  [779] = {x=22.893, y=-17.965, rx=-180, rz=-141.93, shoulder=lefty, elbow=epositive, wrist=wpositive, fatherId=fReference[0]}
  [780] = {x=24.131, y=-18.934, rx=180, rz=-141.938, shoulder=lefty, elbow=epositive, wrist=wpositive, fatherId=fReference[0]}
  [781] = {x=25.369, y=-19.904, rx=-180, rz=-141.947, shoulder=lefty, elbow=epositive, wrist=wpositive, fatherId=fReference[0]}
  [782] = {x=26.607, y=-20.873, rx=-180, rz=-141.956, shoulder=lefty, elbow=epositive, wrist=wpositive, fatherId=fReference[0]}
  [783] = {x=27.846, y=-21.842, rx=-180, rz=-141.965, shoulder=lefty, elbow=epositive, wrist=wpositive, fatherId=fReference[0]}
  [784] = {x=29.084, y=-22.811, rx=-180, rz=-141.975, shoulder=lefty, elbow=epositive, wrist=wpositive, fatherId=fReference[0]}
  [785] = {x=30.323, y=-23.779, rx=180, rz=-141.986, shoulder=lefty, elbow=epositive, wrist=wpositive, fatherId=fReference[0]}
  [786] = {x=31.561, y=-24.748, rx=-180, rz=-141.996, shoulder=lefty, elbow=epositive, wrist=wpositive, fatherId=fReference[0]}
  [787] = {x=32.8, y=-25.716, rx=-180, rz=-142.008, shoulder=lefty, elbow=epositive, wrist=wpositive, fatherId=fReference[0]}
  [788] = {x=34.039, y=-26.683, rx=-180, rz=-142.019, shoulder=lefty, elbow=epositive, wrist=wpositive, fatherId=fReference[0]}
  [789] = {x=35.278, y=-27.651, rx=-180, rz=-142.031, shoulder=lefty, elbow=epositive, wrist=wpositive, fatherId=fReference[0]}
  [790] = {x=36.517, y=-28.618, rx=-180, rz=-142.044, shoulder=lefty, elbow=epositive, wrist=wpositive, fatherId=fReference[0]}
  [791] = {x=37.757, y=-29.585, rx=180, rz=-142.057, shoulder=lefty, elbow=epositive, wrist=wpositive, fatherId=fReference[0]}
  [792] = {x=38.996, y=-30.551, rx=180, rz=-142.07, shoulder=lefty, elbow=epositive, wrist=wpositive, fatherId=fReference[0]}
  [793] = {x=40.236, y=-31.517, rx=180, rz=-142.084, shoulder=lefty, elbow=epositive, wrist=wpositive, fatherId=fReference[0]}
  [794] = {x=41.476, y=-32.483, rx=180, rz=-142.098, shoulder=lefty, elbow=epositive, wrist=wpositive, fatherId=fReference[0]}
  [795] = {x=42.715, y=-33.448, rx=180, rz=-142.113, shoulder=lefty, elbow=epositive, wrist=wpositive, fatherId=fReference[0]}
  [796] = {x=43.956, y=-34.413, rx=-180, rz=-142.128, shoulder=lefty, elbow=epositive, wrist=wpositive, fatherId=fReference[0]}
  [797] = {x=45.196, y=-35.377, rx=180, rz=-142.143, shoulder=lefty, elbow=epositive, wrist=wpositive, fatherId=fReference[0]}
  [798] = {x=46.436, y=-36.342, rx=-180, rz=-142.159, shoulder=lefty, elbow=epositive, wrist=wpositive, fatherId=fReference[0]}
  [799] = {x=47.677, y=-37.305, rx=180, rz=-142.175, shoulder=lefty, elbow=epositive, wrist=wpositive, fatherId=fReference[0]}
  [800] = {x=48.917, y=-38.269, rx=-180, rz=-142.192, shoulder=lefty, elbow=epositive, wrist=wpositive, fatherId=fReference[0]}
  [801] = {x=50.158, y=-39.231, rx=-180, rz=-142.209, shoulder=lefty, elbow=epositive, wrist=wpositive, fatherId=fReference[0]}
  [802] = {x=51.399, y=-40.194, rx=-180, rz=-142.227, shoulder=lefty, elbow=epositive, wrist=wpositive, fatherId=fReference[0]}
  [803] = {x=52.641, y=-41.156, rx=-180, rz=-142.245, shoulder=lefty, elbow=epositive, wrist=wpositive, fatherId=fReference[0]}
  [804] = {x=53.882, y=-42.117, rx=-180, rz=-142.263, shoulder=lefty, elbow=epositive, wrist=wpositive, fatherId=fReference[0]}
  [805] = {x=55.124, y=-43.078, rx=-180, rz=-142.282, shoulder=lefty, elbow=epositive, wrist=wpositive, fatherId=fReference[0]}
  [806] = {x=56.366, y=-44.038, rx=-180, rz=-142.302, shoulder=lefty, elbow=epositive, wrist=wpositive, fatherId=fReference[0]}
  [807] = {x=57.608, y=-44.998, rx=-180, rz=-142.321, shoulder=lefty, elbow=epositive, wrist=wpositive, fatherId=fReference[0]}
  [808] = {x=58.85, y=-45.958, rx=-180, rz=-142.342, shoulder=lefty, elbow=epositive, wrist=wpositive, fatherId=fReference[0]}
  [809] = {x=60.092, y=-46.916, rx=-180, rz=-142.362, shoulder=lefty, elbow=epositive, wrist=wpositive, fatherId=fReference[0]}
  [810] = {x=61.335, y=-47.875, rx=-180, rz=-142.383, shoulder=lefty, elbow=epositive, wrist=wpositive, fatherId=fReference[0]}
  [811] = {x=62.578, y=-48.832, rx=180, rz=-142.405, shoulder=lefty, elbow=epositive, wrist=wpositive, fatherId=fReference[0]}
  [812] = {x=63.821, y=-49.79, rx=-180, rz=-142.427, shoulder=lefty, elbow=epositive, wrist=wpositive, fatherId=fReference[0]}
  [813] = {x=65.064, y=-50.746, rx=180, rz=-142.449, shoulder=lefty, elbow=epositive, wrist=wpositive, fatherId=fReference[0]}
  [814] = {x=66.308, y=-51.702, rx=-180, rz=-142.472, shoulder=lefty, elbow=epositive, wrist=wpositive, fatherId=fReference[0]}
  [815] = {x=67.551, y=-52.657, rx=180, rz=-142.496, shoulder=lefty, elbow=epositive, wrist=wpositive, fatherId=fReference[0]}
  [816] = {x=68.795, y=-53.612, rx=180, rz=-142.519, shoulder=lefty, elbow=epositive, wrist=wpositive, fatherId=fReference[0]}
  [817] = {x=70.04, y=-54.566, rx=180, rz=-142.543, shoulder=lefty, elbow=epositive, wrist=wpositive, fatherId=fReference[0]}
  [818] = {x=71.284, y=-55.519, rx=-180, rz=-142.568, shoulder=lefty, elbow=epositive, wrist=wpositive, fatherId=fReference[0]}
  [819] = {x=72.529, y=-56.472, rx=-180, rz=-142.593, shoulder=lefty, elbow=epositive, wrist=wpositive, fatherId=fReference[0]}
  [820] = {x=73.774, y=-57.424, rx=-180, rz=-142.619, shoulder=lefty, elbow=epositive, wrist=wpositive, fatherId=fReference[0]}
  [821] = {x=75.019, y=-58.376, rx=180, rz=-142.645, shoulder=lefty, elbow=epositive, wrist=wpositive, fatherId=fReference[0]}
  [822] = {x=76.264, y=-59.326, rx=180, rz=-142.671, shoulder=lefty, elbow=epositive, wrist=wpositive, fatherId=fReference[0]}
  [823] = {x=77.51, y=-60.276, rx=180, rz=-142.698, shoulder=lefty, elbow=epositive, wrist=wpositive, fatherId=fReference[0]}
  [824] = {x=78.756, y=-61.226, rx=-180, rz=-142.725, shoulder=lefty, elbow=epositive, wrist=wpositive, fatherId=fReference[0]}
  [825] = {x=80.002, y=-62.174, rx=-180, rz=-142.753, shoulder=lefty, elbow=epositive, wrist=wpositive, fatherId=fReference[0]}
  [826] = {x=81.249, y=-63.122, rx=-180, rz=-142.781, shoulder=lefty, elbow=epositive, wrist=wpositive, fatherId=fReference[0]}
  [827] = {x=82.496, y=-64.069, rx=-180, rz=-142.81, shoulder=lefty, elbow=epositive, wrist=wpositive, fatherId=fReference[0]}
  [828] = {x=83.743, y=-65.015, rx=180, rz=-142.839, shoulder=lefty, elbow=epositive, wrist=wpositive, fatherId=fReference[0]}
  [829] = {x=84.99, y=-65.961, rx=180, rz=-142.868, shoulder=lefty, elbow=epositive, wrist=wpositive, fatherId=fReference[0]}
  [830] = {x=86.238, y=-66.905, rx=-180, rz=-142.898, shoulder=lefty, elbow=epositive, wrist=wpositive, fatherId=fReference[0]}
  [831] = {x=87.486, y=-67.849, rx=-180, rz=-142.929, shoulder=lefty, elbow=epositive, wrist=wpositive, fatherId=fReference[0]}
  [832] = {x=88.734, y=-68.792, rx=-180, rz=-142.96, shoulder=lefty, elbow=epositive, wrist=wpositive, fatherId=fReference[0]}
  [833] = {x=89.982, y=-69.734, rx=-180, rz=-142.991, shoulder=lefty, elbow=epositive, wrist=wpositive, fatherId=fReference[0]}
  [834] = {x=91.231, y=-70.676, rx=-180, rz=-143.023, shoulder=lefty, elbow=epositive, wrist=wpositive, fatherId=fReference[0]}
  [835] = {x=92.48, y=-71.616, rx=-180, rz=-143.055, shoulder=lefty, elbow=epositive, wrist=wpositive, fatherId=fReference[0]}
  [836] = {x=93.73, y=-72.556, rx=-180, rz=-143.088, shoulder=lefty, elbow=epositive, wrist=wpositive, fatherId=fReference[0]}
  [837] = {x=94.979, y=-73.495, rx=-180, rz=-143.121, shoulder=lefty, elbow=epositive, wrist=wpositive, fatherId=fReference[0]}
  [838] = {x=96.23, y=-74.432, rx=-180, rz=-143.155, shoulder=lefty, elbow=epositive, wrist=wpositive, fatherId=fReference[0]}
  [839] = {x=97.48, y=-75.369, rx=-180, rz=-143.189, shoulder=lefty, elbow=epositive, wrist=wpositive, fatherId=fReference[0]}
  [840] = {x=98.731, y=-76.305, rx=-180, rz=-143.224, shoulder=lefty, elbow=epositive, wrist=wpositive, fatherId=fReference[0]}
  [841] = {x=99.982, y=-77.24, rx=180, rz=-143.259, shoulder=lefty, elbow=epositive, wrist=wpositive, fatherId=fReference[0]}
  [842] = {x=101.233, y=-78.175, rx=-180, rz=-143.294, shoulder=lefty, elbow=epositive, wrist=wpositive, fatherId=fReference[0]}
  [843] = {x=102.485, y=-79.108, rx=-180, rz=-143.33, shoulder=lefty, elbow=epositive, wrist=wpositive, fatherId=fReference[0]}
  [844] = {x=103.737, y=-80.04, rx=-180, rz=-143.367, shoulder=lefty, elbow=epositive, wrist=wpositive, fatherId=fReference[0]}
  [845] = {x=104.989, y=-80.971, rx=-180, rz=-143.404, shoulder=lefty, elbow=epositive, wrist=wpositive, fatherId=fReference[0]}
  [846] = {x=106.242, y=-81.901, rx=-180, rz=-143.441, shoulder=lefty, elbow=epositive, wrist=wpositive, fatherId=fReference[0]}
  [847] = {x=107.495, y=-82.831, rx=-180, rz=-143.479, shoulder=lefty, elbow=epositive, wrist=wpositive, fatherId=fReference[0]}
  [848] = {x=108.748, y=-83.759, rx=-180, rz=-143.517, shoulder=lefty, elbow=epositive, wrist=wpositive, fatherId=fReference[0]}
  [849] = {x=110.002, y=-84.686, rx=-180, rz=-143.556, shoulder=lefty, elbow=epositive, wrist=wpositive, fatherId=fReference[0]}
  [850] = {x=111.256, y=-85.612, rx=-180, rz=-143.596, shoulder=lefty, elbow=epositive, wrist=wpositive, fatherId=fReference[0]}
  [851] = {x=112.511, y=-86.537, rx=-180, rz=-143.635, shoulder=lefty, elbow=epositive, wrist=wpositive, fatherId=fReference[0]}
  [852] = {x=113.766, y=-87.461, rx=180, rz=-143.676, shoulder=lefty, elbow=epositive, wrist=wpositive, fatherId=fReference[0]}
  [853] = {x=115.021, y=-88.384, rx=180, rz=-143.716, shoulder=lefty, elbow=epositive, wrist=wpositive, fatherId=fReference[0]}
  [854] = {x=116.277, y=-89.306, rx=-180, rz=-143.758, shoulder=lefty, elbow=epositive, wrist=wpositive, fatherId=fReference[0]}
  [855] = {x=117.533, y=-90.227, rx=-180, rz=-143.799, shoulder=lefty, elbow=epositive, wrist=wpositive, fatherId=fReference[0]}
  [856] = {x=118.789, y=-91.146, rx=180, rz=-143.842, shoulder=lefty, elbow=epositive, wrist=wpositive, fatherId=fReference[0]}
  [857] = {x=120.046, y=-92.065, rx=-180, rz=-143.884, shoulder=lefty, elbow=epositive, wrist=wpositive, fatherId=fReference[0]}
  [858] = {x=121.304, y=-92.982, rx=-180, rz=-143.927, shoulder=lefty, elbow=epositive, wrist=wpositive, fatherId=fReference[0]}
  [859] = {x=122.561, y=-93.898, rx=180, rz=-143.971, shoulder=lefty, elbow=epositive, wrist=wpositive, fatherId=fReference[0]}
  [860] = {x=123.819, y=-94.813, rx=180, rz=-144.015, shoulder=lefty, elbow=epositive, wrist=wpositive, fatherId=fReference[0]}
  [861] = {x=125.078, y=-95.727, rx=-180, rz=-144.06, shoulder=lefty, elbow=epositive, wrist=wpositive, fatherId=fReference[0]}
  [862] = {x=126.337, y=-96.64, rx=-180, rz=-144.105, shoulder=lefty, elbow=epositive, wrist=wpositive, fatherId=fReference[0]}
  [863] = {x=127.596, y=-97.551, rx=-180, rz=-144.151, shoulder=lefty, elbow=epositive, wrist=wpositive, fatherId=fReference[0]}
  [864] = {x=128.856, y=-98.461, rx=180, rz=-144.197, shoulder=lefty, elbow=epositive, wrist=wpositive, fatherId=fReference[0]}
  [865] = {x=130.116, y=-99.37, rx=180, rz=-144.243, shoulder=lefty, elbow=epositive, wrist=wpositive, fatherId=fReference[0]}
  [866] = {x=131.376, y=-100.278, rx=-180, rz=-144.291, shoulder=lefty, elbow=epositive, wrist=wpositive, fatherId=fReference[0]}
  [867] = {x=132.637, y=-101.185, rx=180, rz=-144.338, shoulder=lefty, elbow=epositive, wrist=wpositive, fatherId=fReference[0]}
  [868] = {x=133.899, y=-102.09, rx=180, rz=-144.386, shoulder=lefty, elbow=epositive, wrist=wpositive, fatherId=fReference[0]}
  [869] = {x=135.161, y=-102.994, rx=180, rz=-144.435, shoulder=lefty, elbow=epositive, wrist=wpositive, fatherId=fReference[0]}
  [870] = {x=136.423, y=-103.896, rx=-180, rz=-144.484, shoulder=lefty, elbow=epositive, wrist=wpositive, fatherId=fReference[0]}
  [871] = {x=137.686, y=-104.798, rx=-180, rz=-144.534, shoulder=lefty, elbow=epositive, wrist=wpositive, fatherId=fReference[0]}
  [872] = {x=138.949, y=-105.698, rx=-180, rz=-144.584, shoulder=lefty, elbow=epositive, wrist=wpositive, fatherId=fReference[0]}
  [873] = {x=140.213, y=-106.596, rx=-180, rz=-144.634, shoulder=lefty, elbow=epositive, wrist=wpositive, fatherId=fReference[0]}
  [874] = {x=141.477, y=-107.494, rx=-180, rz=-144.686, shoulder=lefty, elbow=epositive, wrist=wpositive, fatherId=fReference[0]}
  [875] = {x=142.742, y=-108.389, rx=-180, rz=-144.737, shoulder=lefty, elbow=epositive, wrist=wpositive, fatherId=fReference[0]}
  [876] = {x=144.007, y=-109.284, rx=180, rz=-144.789, shoulder=lefty, elbow=epositive, wrist=wpositive, fatherId=fReference[0]}
  [877] = {x=145.273, y=-110.177, rx=180, rz=-144.842, shoulder=lefty, elbow=epositive, wrist=wpositive, fatherId=fReference[0]}
  [878] = {x=146.539, y=-111.069, rx=180, rz=-144.895, shoulder=lefty, elbow=epositive, wrist=wpositive, fatherId=fReference[0]}
  [879] = {x=147.806, y=-111.959, rx=180, rz=-144.949, shoulder=lefty, elbow=epositive, wrist=wpositive, fatherId=fReference[0]}
  [880] = {x=149.073, y=-112.848, rx=-180, rz=-145.003, shoulder=lefty, elbow=epositive, wrist=wpositive, fatherId=fReference[0]}
  [881] = {x=150.34, y=-113.736, rx=180, rz=-145.058, shoulder=lefty, elbow=epositive, wrist=wpositive, fatherId=fReference[0]}
  [882] = {x=151.608, y=-114.622, rx=180, rz=-145.113, shoulder=lefty, elbow=epositive, wrist=wpositive, fatherId=fReference[0]}
  [883] = {x=152.877, y=-115.506, rx=-180, rz=-145.169, shoulder=lefty, elbow=epositive, wrist=wpositive, fatherId=fReference[0]}
  [884] = {x=154.146, y=-116.389, rx=-180, rz=-145.225, shoulder=lefty, elbow=epositive, wrist=wpositive, fatherId=fReference[0]}
  [885] = {x=155.416, y=-117.271, rx=-180, rz=-145.282, shoulder=lefty, elbow=epositive, wrist=wpositive, fatherId=fReference[0]}
  [886] = {x=156.686, y=-118.151, rx=-180, rz=-145.34, shoulder=lefty, elbow=epositive, wrist=wpositive, fatherId=fReference[0]}
  [887] = {x=157.957, y=-119.03, rx=-180, rz=-145.398, shoulder=lefty, elbow=epositive, wrist=wpositive, fatherId=fReference[0]}
  [888] = {x=159.228, y=-119.907, rx=-180, rz=-145.456, shoulder=lefty, elbow=epositive, wrist=wpositive, fatherId=fReference[0]}
  [889] = {x=160.5, y=-120.782, rx=180, rz=-145.515, shoulder=lefty, elbow=epositive, wrist=wpositive, fatherId=fReference[0]}
  [890] = {x=161.772, y=-121.656, rx=180, rz=-145.575, shoulder=lefty, elbow=epositive, wrist=wpositive, fatherId=fReference[0]}
  [891] = {x=163.045, y=-122.529, rx=-180, rz=-145.635, shoulder=lefty, elbow=epositive, wrist=wpositive, fatherId=fReference[0]}
  [892] = {x=164.319, y=-123.4, rx=-180, rz=-145.695, shoulder=lefty, elbow=epositive, wrist=wpositive, fatherId=fReference[0]}
  [893] = {x=165.593, y=-124.269, rx=-180, rz=-145.756, shoulder=lefty, elbow=epositive, wrist=wpositive, fatherId=fReference[0]}
  [894] = {x=166.867, y=-125.136, rx=180, rz=-145.818, shoulder=lefty, elbow=epositive, wrist=wpositive, fatherId=fReference[0]}
  [895] = {x=168.142, y=-126.002, rx=-180, rz=-145.88, shoulder=lefty, elbow=epositive, wrist=wpositive, fatherId=fReference[0]}
  [896] = {x=169.418, y=-126.867, rx=-180, rz=-145.943, shoulder=lefty, elbow=epositive, wrist=wpositive, fatherId=fReference[0]}
  [897] = {x=170.695, y=-127.73, rx=-180, rz=-146.006, shoulder=lefty, elbow=epositive, wrist=wpositive, fatherId=fReference[0]}
  [898] = {x=171.971, y=-128.591, rx=180, rz=-146.07, shoulder=lefty, elbow=epositive, wrist=wpositive, fatherId=fReference[0]}
  [899] = {x=173.249, y=-129.45, rx=180, rz=-146.135, shoulder=lefty, elbow=epositive, wrist=wpositive, fatherId=fReference[0]}
  [900] = {x=174.527, y=-130.308, rx=-180, rz=-146.2, shoulder=lefty, elbow=epositive, wrist=wpositive, fatherId=fReference[0]}
  [901] = {x=175.806, y=-131.164, rx=-180, rz=-146.265, shoulder=lefty, elbow=epositive, wrist=wpositive, fatherId=fReference[0]}
  [902] = {x=177.085, y=-132.018, rx=-180, rz=-146.331, shoulder=lefty, elbow=epositive, wrist=wpositive, fatherId=fReference[0]}
  [903] = {x=178.365, y=-132.871, rx=180, rz=-146.398, shoulder=lefty, elbow=epositive, wrist=wpositive, fatherId=fReference[0]}
  [904] = {x=179.645, y=-133.721, rx=-180, rz=-146.465, shoulder=lefty, elbow=epositive, wrist=wpositive, fatherId=fReference[0]}
  [905] = {x=180.927, y=-134.571, rx=-180, rz=-146.533, shoulder=lefty, elbow=epositive, wrist=wpositive, fatherId=fReference[0]}
  [906] = {x=182.208, y=-135.418, rx=-180, rz=-146.601, shoulder=lefty, elbow=epositive, wrist=wpositive, fatherId=fReference[0]}
  [907] = {x=183.491, y=-136.263, rx=-180, rz=-146.67, shoulder=lefty, elbow=epositive, wrist=wpositive, fatherId=fReference[0]}
  [908] = {x=184.774, y=-137.107, rx=-180, rz=-146.74, shoulder=lefty, elbow=epositive, wrist=wpositive, fatherId=fReference[0]}
  [909] = {x=186.057, y=-137.949, rx=-180, rz=-146.81, shoulder=lefty, elbow=epositive, wrist=wpositive, fatherId=fReference[0]}
  [910] = {x=187.341, y=-138.789, rx=-180, rz=-146.881, shoulder=lefty, elbow=epositive, wrist=wpositive, fatherId=fReference[0]}
  [911] = {x=188.626, y=-139.627, rx=-180, rz=-146.952, shoulder=lefty, elbow=epositive, wrist=wpositive, fatherId=fReference[0]}
  [912] = {x=189.912, y=-140.464, rx=-180, rz=-147.024, shoulder=lefty, elbow=epositive, wrist=wpositive, fatherId=fReference[0]}
  [913] = {x=191.198, y=-141.298, rx=-180, rz=-147.096, shoulder=lefty, elbow=epositive, wrist=wpositive, fatherId=fReference[0]}
  [914] = {x=192.485, y=-142.131, rx=-180, rz=-147.169, shoulder=lefty, elbow=epositive, wrist=wpositive, fatherId=fReference[0]}
  [915] = {x=193.772, y=-142.961, rx=-180, rz=-147.243, shoulder=lefty, elbow=epositive, wrist=wpositive, fatherId=fReference[0]}
  [916] = {x=195.06, y=-143.79, rx=-180, rz=-147.317, shoulder=lefty, elbow=epositive, wrist=wpositive, fatherId=fReference[0]}
  [917] = {x=196.349, y=-144.617, rx=180, rz=-147.392, shoulder=lefty, elbow=epositive, wrist=wpositive, fatherId=fReference[0]}
  [918] = {x=197.639, y=-145.442, rx=-180, rz=-147.467, shoulder=lefty, elbow=epositive, wrist=wpositive, fatherId=fReference[0]}
  [919] = {x=198.929, y=-146.265, rx=-180, rz=-147.543, shoulder=lefty, elbow=epositive, wrist=wpositive, fatherId=fReference[0]}
  [920] = {x=200.219, y=-147.086, rx=-180, rz=-147.619, shoulder=lefty, elbow=epositive, wrist=wpositive, fatherId=fReference[0]}
  [921] = {x=201.511, y=-147.905, rx=-180, rz=-147.697, shoulder=lefty, elbow=epositive, wrist=wpositive, fatherId=fReference[0]}
  [922] = {x=202.803, y=-148.722, rx=180, rz=-147.774, shoulder=lefty, elbow=epositive, wrist=wpositive, fatherId=fReference[0]}
  [923] = {x=204.096, y=-149.536, rx=-180, rz=-147.853, shoulder=lefty, elbow=epositive, wrist=wpositive, fatherId=fReference[0]}
  [924] = {x=205.389, y=-150.349, rx=-180, rz=-147.931, shoulder=lefty, elbow=epositive, wrist=wpositive, fatherId=fReference[0]}
  [925] = {x=206.683, y=-151.16, rx=-180, rz=-148.011, shoulder=lefty, elbow=epositive, wrist=wpositive, fatherId=fReference[0]}
  [926] = {x=207.978, y=-151.969, rx=-180, rz=-148.091, shoulder=lefty, elbow=epositive, wrist=wpositive, fatherId=fReference[0]}
  [927] = {x=209.273, y=-152.775, rx=-180, rz=-148.172, shoulder=lefty, elbow=epositive, wrist=wpositive, fatherId=fReference[0]}
  [928] = {x=210.569, y=-153.58, rx=-180, rz=-148.253, shoulder=lefty, elbow=epositive, wrist=wpositive, fatherId=fReference[0]}
  [929] = {x=211.866, y=-154.382, rx=-180, rz=-148.335, shoulder=lefty, elbow=epositive, wrist=wpositive, fatherId=fReference[0]}
  [930] = {x=213.164, y=-155.183, rx=-180, rz=-148.418, shoulder=lefty, elbow=epositive, wrist=wpositive, fatherId=fReference[0]}
  [931] = {x=214.462, y=-155.981, rx=180, rz=-148.501, shoulder=lefty, elbow=epositive, wrist=wpositive, fatherId=fReference[0]}
  [932] = {x=215.761, y=-156.777, rx=-180, rz=-148.585, shoulder=lefty, elbow=epositive, wrist=wpositive, fatherId=fReference[0]}
  [933] = {x=217.06, y=-157.57, rx=-180, rz=-148.669, shoulder=lefty, elbow=epositive, wrist=wpositive, fatherId=fReference[0]}
  [934] = {x=218.361, y=-158.362, rx=-180, rz=-148.754, shoulder=lefty, elbow=epositive, wrist=wpositive, fatherId=fReference[0]}
  [935] = {x=219.662, y=-159.151, rx=-180, rz=-148.84, shoulder=lefty, elbow=epositive, wrist=wpositive, fatherId=fReference[0]}
  [936] = {x=220.963, y=-159.938, rx=-180, rz=-148.926, shoulder=lefty, elbow=epositive, wrist=wpositive, fatherId=fReference[0]}
  [937] = {x=222.266, y=-160.723, rx=180, rz=-149.013, shoulder=lefty, elbow=epositive, wrist=wpositive, fatherId=fReference[0]}
  [938] = {x=223.569, y=-161.506, rx=-180, rz=-149.101, shoulder=lefty, elbow=epositive, wrist=wpositive, fatherId=fReference[0]}
  [939] = {x=224.872, y=-162.286, rx=-180, rz=-149.189, shoulder=lefty, elbow=epositive, wrist=wpositive, fatherId=fReference[0]}
  [940] = {x=226.177, y=-163.064, rx=-180, rz=-149.278, shoulder=lefty, elbow=epositive, wrist=wpositive, fatherId=fReference[0]}
  [941] = {x=227.482, y=-163.84, rx=-180, rz=-149.367, shoulder=lefty, elbow=epositive, wrist=wpositive, fatherId=fReference[0]}
  [942] = {x=228.788, y=-164.613, rx=-180, rz=-149.458, shoulder=lefty, elbow=epositive, wrist=wpositive, fatherId=fReference[0]}
  [943] = {x=230.095, y=-165.384, rx=-180, rz=-149.548, shoulder=lefty, elbow=epositive, wrist=wpositive, fatherId=fReference[0]}
  [944] = {x=231.402, y=-166.152, rx=-180, rz=-149.64, shoulder=lefty, elbow=epositive, wrist=wpositive, fatherId=fReference[0]}
  [945] = {x=232.71, y=-166.919, rx=-180, rz=-149.732, shoulder=lefty, elbow=epositive, wrist=wpositive, fatherId=fReference[0]}
  [946] = {x=234.019, y=-167.682, rx=-180, rz=-149.824, shoulder=lefty, elbow=epositive, wrist=wpositive, fatherId=fReference[0]}
  [947] = {x=235.328, y=-168.444, rx=-180, rz=-149.918, shoulder=lefty, elbow=epositive, wrist=wpositive, fatherId=fReference[0]}
  [948] = {x=236.638, y=-169.203, rx=180, rz=-150.012, shoulder=lefty, elbow=epositive, wrist=wpositive, fatherId=fReference[0]}
  [949] = {x=237.949, y=-169.959, rx=-180, rz=-150.106, shoulder=lefty, elbow=epositive, wrist=wpositive, fatherId=fReference[0]}
  [950] = {x=239.261, y=-170.713, rx=-180, rz=-150.202, shoulder=lefty, elbow=epositive, wrist=wpositive, fatherId=fReference[0]}
  [951] = {x=240.573, y=-171.465, rx=180, rz=-150.298, shoulder=lefty, elbow=epositive, wrist=wpositive, fatherId=fReference[0]}
  [952] = {x=241.886, y=-172.214, rx=-180, rz=-150.394, shoulder=lefty, elbow=epositive, wrist=wpositive, fatherId=fReference[0]}
  [953] = {x=243.2, y=-172.96, rx=-180, rz=-150.491, shoulder=lefty, elbow=epositive, wrist=wpositive, fatherId=fReference[0]}
  [954] = {x=244.514, y=-173.704, rx=-180, rz=-150.589, shoulder=lefty, elbow=epositive, wrist=wpositive, fatherId=fReference[0]}
  [955] = {x=245.83, y=-174.446, rx=180, rz=-150.688, shoulder=lefty, elbow=epositive, wrist=wpositive, fatherId=fReference[0]}
  [956] = {x=247.146, y=-175.184, rx=-180, rz=-150.787, shoulder=lefty, elbow=epositive, wrist=wpositive, fatherId=fReference[0]}
  [957] = {x=248.462, y=-175.921, rx=-180, rz=-150.887, shoulder=lefty, elbow=epositive, wrist=wpositive, fatherId=fReference[0]}
  [958] = {x=249.78, y=-176.654, rx=-180, rz=-150.988, shoulder=lefty, elbow=epositive, wrist=wpositive, fatherId=fReference[0]}
  [959] = {x=251.098, y=-177.385, rx=180, rz=-151.089, shoulder=lefty, elbow=epositive, wrist=wpositive, fatherId=fReference[0]}
  [960] = {x=252.417, y=-178.114, rx=-180, rz=-151.191, shoulder=lefty, elbow=epositive, wrist=wpositive, fatherId=fReference[0]}
  [961] = {x=253.736, y=-178.839, rx=-180, rz=-151.293, shoulder=lefty, elbow=epositive, wrist=wpositive, fatherId=fReference[0]}
  [962] = {x=255.056, y=-179.562, rx=-180, rz=-151.397, shoulder=lefty, elbow=epositive, wrist=wpositive, fatherId=fReference[0]}
  [963] = {x=256.378, y=-180.283, rx=-180, rz=-151.501, shoulder=lefty, elbow=epositive, wrist=wpositive, fatherId=fReference[0]}
  [964] = {x=257.699, y=-181, rx=-180, rz=-151.605, shoulder=lefty, elbow=epositive, wrist=wpositive, fatherId=fReference[0]}
  [965] = {x=259.022, y=-181.715, rx=-180, rz=-151.711, shoulder=lefty, elbow=epositive, wrist=wpositive, fatherId=fReference[0]}
  [966] = {x=260.345, y=-182.427, rx=-180, rz=-151.817, shoulder=lefty, elbow=epositive, wrist=wpositive, fatherId=fReference[0]}
  [967] = {x=261.669, y=-183.137, rx=-180, rz=-151.923, shoulder=lefty, elbow=epositive, wrist=wpositive, fatherId=fReference[0]}
  [968] = {x=262.994, y=-183.843, rx=-180, rz=-152.031, shoulder=lefty, elbow=epositive, wrist=wpositive, fatherId=fReference[0]}
  [969] = {x=264.319, y=-184.547, rx=-180, rz=-152.139, shoulder=lefty, elbow=epositive, wrist=wpositive, fatherId=fReference[0]}
  [970] = {x=265.645, y=-185.248, rx=180, rz=-152.247, shoulder=lefty, elbow=epositive, wrist=wpositive, fatherId=fReference[0]}
  [971] = {x=266.972, y=-185.946, rx=-180, rz=-152.357, shoulder=lefty, elbow=epositive, wrist=wpositive, fatherId=fReference[0]}
  [972] = {x=268.3, y=-186.642, rx=-180, rz=-152.467, shoulder=lefty, elbow=epositive, wrist=wpositive, fatherId=fReference[0]}
  [973] = {x=269.628, y=-187.334, rx=-180, rz=-152.578, shoulder=lefty, elbow=epositive, wrist=wpositive, fatherId=fReference[0]}
  [974] = {x=270.957, y=-188.024, rx=-180, rz=-152.689, shoulder=lefty, elbow=epositive, wrist=wpositive, fatherId=fReference[0]}
  [975] = {x=272.287, y=-188.711, rx=-180, rz=-152.801, shoulder=lefty, elbow=epositive, wrist=wpositive, fatherId=fReference[0]}
  [976] = {x=273.617, y=-189.394, rx=-180, rz=-152.914, shoulder=lefty, elbow=epositive, wrist=wpositive, fatherId=fReference[0]}
  [977] = {x=274.948, y=-190.075, rx=-180, rz=-153.028, shoulder=lefty, elbow=epositive, wrist=wpositive, fatherId=fReference[0]}
  [978] = {x=276.28, y=-190.753, rx=-180, rz=-153.142, shoulder=lefty, elbow=epositive, wrist=wpositive, fatherId=fReference[0]}
  [979] = {x=277.613, y=-191.428, rx=-180, rz=-153.257, shoulder=lefty, elbow=epositive, wrist=wpositive, fatherId=fReference[0]}
  [980] = {x=278.947, y=-192.1, rx=180, rz=-153.372, shoulder=lefty, elbow=epositive, wrist=wpositive, fatherId=fReference[0]}
  [981] = {x=280.281, y=-192.769, rx=180, rz=-153.489, shoulder=lefty, elbow=epositive, wrist=wpositive, fatherId=fReference[0]}
  [982] = {x=281.616, y=-193.435, rx=180, rz=-153.606, shoulder=lefty, elbow=epositive, wrist=wpositive, fatherId=fReference[0]}
  [983] = {x=282.951, y=-194.097, rx=180, rz=-153.724, shoulder=lefty, elbow=epositive, wrist=wpositive, fatherId=fReference[0]}
  [984] = {x=284.288, y=-194.757, rx=180, rz=-153.842, shoulder=lefty, elbow=epositive, wrist=wpositive, fatherId=fReference[0]}
  [985] = {x=285.625, y=-195.414, rx=-180, rz=-153.961, shoulder=lefty, elbow=epositive, wrist=wpositive, fatherId=fReference[0]}
  [986] = {x=286.963, y=-196.068, rx=180, rz=-154.081, shoulder=lefty, elbow=epositive, wrist=wpositive, fatherId=fReference[0]}
  [987] = {x=288.301, y=-196.718, rx=180, rz=-154.202, shoulder=lefty, elbow=epositive, wrist=wpositive, fatherId=fReference[0]}
  [988] = {x=289.64, y=-197.365, rx=-180, rz=-154.323, shoulder=lefty, elbow=epositive, wrist=wpositive, fatherId=fReference[0]}
  [989] = {x=290.98, y=-198.01, rx=180, rz=-154.445, shoulder=lefty, elbow=epositive, wrist=wpositive, fatherId=fReference[0]}
  [990] = {x=292.321, y=-198.651, rx=180, rz=-154.568, shoulder=lefty, elbow=epositive, wrist=wpositive, fatherId=fReference[0]}
  [991] = {x=293.663, y=-199.289, rx=180, rz=-154.691, shoulder=lefty, elbow=epositive, wrist=wpositive, fatherId=fReference[0]}
  [992] = {x=295.005, y=-199.923, rx=180, rz=-154.815, shoulder=lefty, elbow=epositive, wrist=wpositive, fatherId=fReference[0]}
  [993] = {x=296.348, y=-200.555, rx=180, rz=-154.94, shoulder=lefty, elbow=epositive, wrist=wpositive, fatherId=fReference[0]}
  [994] = {x=297.691, y=-201.183, rx=-180, rz=-155.066, shoulder=lefty, elbow=epositive, wrist=wpositive, fatherId=fReference[0]}
  [995] = {x=299.036, y=-201.808, rx=-180, rz=-155.192, shoulder=lefty, elbow=epositive, wrist=wpositive, fatherId=fReference[0]}
  [996] = {x=300.381, y=-202.43, rx=180, rz=-155.319, shoulder=lefty, elbow=epositive, wrist=wpositive, fatherId=fReference[0]}
  [997] = {x=301.727, y=-203.048, rx=-180, rz=-155.447, shoulder=lefty, elbow=epositive, wrist=wpositive, fatherId=fReference[0]}
  [998] = {x=303.073, y=-203.663, rx=-180, rz=-155.575, shoulder=lefty, elbow=epositive, wrist=wpositive, fatherId=fReference[0]}
  [999] = {x=304.421, y=-204.275, rx=-180, rz=-155.705, shoulder=lefty, elbow=epositive, wrist=wpositive, fatherId=fReference[0]}
  [1000] = {x=305.769, y=-204.884, rx=-180, rz=-155.835, shoulder=lefty, elbow=epositive, wrist=wpositive, fatherId=fReference[0]}
  [1001] = {x=307.117, y=-205.489, rx=-180, rz=-155.965, shoulder=lefty, elbow=epositive, wrist=wpositive, fatherId=fReference[0]}
  [1002] = {x=308.467, y=-206.091, rx=-180, rz=-156.097, shoulder=lefty, elbow=epositive, wrist=wpositive, fatherId=fReference[0]}
  [1003] = {x=309.817, y=-206.689, rx=-180, rz=-156.229, shoulder=lefty, elbow=epositive, wrist=wpositive, fatherId=fReference[0]}
  [1004] = {x=311.168, y=-207.284, rx=180, rz=-156.361, shoulder=lefty, elbow=epositive, wrist=wpositive, fatherId=fReference[0]}
  [1005] = {x=312.519, y=-207.876, rx=-180, rz=-156.495, shoulder=lefty, elbow=epositive, wrist=wpositive, fatherId=fReference[0]}
  [1006] = {x=313.872, y=-208.464, rx=180, rz=-156.629, shoulder=lefty, elbow=epositive, wrist=wpositive, fatherId=fReference[0]}
  [1007] = {x=315.225, y=-209.049, rx=-180, rz=-156.764, shoulder=lefty, elbow=epositive, wrist=wpositive, fatherId=fReference[0]}
  [1008] = {x=316.579, y=-209.63, rx=-180, rz=-156.9, shoulder=lefty, elbow=epositive, wrist=wpositive, fatherId=fReference[0]}
  [1009] = {x=317.933, y=-210.208, rx=180, rz=-157.036, shoulder=lefty, elbow=epositive, wrist=wpositive, fatherId=fReference[0]}
  [1010] = {x=319.288, y=-210.782, rx=-180, rz=-157.173, shoulder=lefty, elbow=epositive, wrist=wpositive, fatherId=fReference[0]}
  [1011] = {x=320.644, y=-211.353, rx=180, rz=-157.311, shoulder=lefty, elbow=epositive, wrist=wpositive, fatherId=fReference[0]}
  [1012] = {x=322.001, y=-211.92, rx=-180, rz=-157.45, shoulder=lefty, elbow=epositive, wrist=wpositive, fatherId=fReference[0]}
  [1013] = {x=323.358, y=-212.483, rx=-180, rz=-157.589, shoulder=lefty, elbow=epositive, wrist=wpositive, fatherId=fReference[0]}
  [1014] = {x=324.716, y=-213.044, rx=-180, rz=-157.729, shoulder=lefty, elbow=epositive, wrist=wpositive, fatherId=fReference[0]}
  [1015] = {x=326.075, y=-213.6, rx=180, rz=-157.87, shoulder=lefty, elbow=epositive, wrist=wpositive, fatherId=fReference[0]}
  [1016] = {x=327.435, y=-214.153, rx=-180, rz=-158.011, shoulder=lefty, elbow=epositive, wrist=wpositive, fatherId=fReference[0]}
  [1017] = {x=328.795, y=-214.702, rx=-180, rz=-158.153, shoulder=lefty, elbow=epositive, wrist=wpositive, fatherId=fReference[0]}
  [1018] = {x=330.156, y=-215.248, rx=-180, rz=-158.296, shoulder=lefty, elbow=epositive, wrist=wpositive, fatherId=fReference[0]}
  [1019] = {x=331.517, y=-215.79, rx=-180, rz=-158.44, shoulder=lefty, elbow=epositive, wrist=wpositive, fatherId=fReference[0]}
  [1020] = {x=332.88, y=-216.328, rx=180, rz=-158.584, shoulder=lefty, elbow=epositive, wrist=wpositive, fatherId=fReference[0]}
  [1021] = {x=334.243, y=-216.863, rx=180, rz=-158.729, shoulder=lefty, elbow=epositive, wrist=wpositive, fatherId=fReference[0]}
  [1022] = {x=335.607, y=-217.394, rx=180, rz=-158.875, shoulder=lefty, elbow=epositive, wrist=wpositive, fatherId=fReference[0]}
  [1023] = {x=336.971, y=-217.921, rx=-180, rz=-159.022, shoulder=lefty, elbow=epositive, wrist=wpositive, fatherId=fReference[0]}
  [1024] = {x=338.336, y=-218.444, rx=-180, rz=-159.169, shoulder=lefty, elbow=epositive, wrist=wpositive, fatherId=fReference[0]}
  [1025] = {x=339.702, y=-218.964, rx=-180, rz=-159.317, shoulder=lefty, elbow=epositive, wrist=wpositive, fatherId=fReference[0]}
  [1026] = {x=341.069, y=-219.48, rx=-180, rz=-159.465, shoulder=lefty, elbow=epositive, wrist=wpositive, fatherId=fReference[0]}
  [1027] = {x=342.436, y=-219.992, rx=-180, rz=-159.615, shoulder=lefty, elbow=epositive, wrist=wpositive, fatherId=fReference[0]}
  [1028] = {x=343.804, y=-220.5, rx=180, rz=-159.765, shoulder=lefty, elbow=epositive, wrist=wpositive, fatherId=fReference[0]}
  [1029] = {x=345.173, y=-221.005, rx=-180, rz=-159.916, shoulder=lefty, elbow=epositive, wrist=wpositive, fatherId=fReference[0]}
  [1030] = {x=346.542, y=-221.506, rx=-180, rz=-160.067, shoulder=lefty, elbow=epositive, wrist=wpositive, fatherId=fReference[0]}
  [1031] = {x=347.912, y=-222.002, rx=-180, rz=-160.219, shoulder=lefty, elbow=epositive, wrist=wpositive, fatherId=fReference[0]}
  [1032] = {x=349.283, y=-222.495, rx=180, rz=-160.372, shoulder=lefty, elbow=epositive, wrist=wpositive, fatherId=fReference[0]}
  [1033] = {x=350.655, y=-222.985, rx=-180, rz=-160.526, shoulder=lefty, elbow=epositive, wrist=wpositive, fatherId=fReference[0]}
  [1034] = {x=352.027, y=-223.47, rx=-180, rz=-160.68, shoulder=lefty, elbow=epositive, wrist=wpositive, fatherId=fReference[0]}
  [1035] = {x=353.4, y=-223.951, rx=-180, rz=-160.835, shoulder=lefty, elbow=epositive, wrist=wpositive, fatherId=fReference[0]}
  [1036] = {x=354.773, y=-224.429, rx=-180, rz=-160.991, shoulder=lefty, elbow=epositive, wrist=wpositive, fatherId=fReference[0]}
  [1037] = {x=356.148, y=-224.902, rx=-180, rz=-161.147, shoulder=lefty, elbow=epositive, wrist=wpositive, fatherId=fReference[0]}
  [1038] = {x=357.523, y=-225.371, rx=-180, rz=-161.304, shoulder=lefty, elbow=epositive, wrist=wpositive, fatherId=fReference[0]}
  [1039] = {x=358.898, y=-225.837, rx=-180, rz=-161.462, shoulder=lefty, elbow=epositive, wrist=wpositive, fatherId=fReference[0]}
  [1040] = {x=360.275, y=-226.298, rx=180, rz=-161.621, shoulder=lefty, elbow=epositive, wrist=wpositive, fatherId=fReference[0]}
  [1041] = {x=361.652, y=-226.756, rx=-180, rz=-161.78, shoulder=lefty, elbow=epositive, wrist=wpositive, fatherId=fReference[0]}
  [1042] = {x=363.029, y=-227.209, rx=-180, rz=-161.94, shoulder=lefty, elbow=epositive, wrist=wpositive, fatherId=fReference[0]}
  [1043] = {x=364.407, y=-227.659, rx=-180, rz=-162.1, shoulder=lefty, elbow=epositive, wrist=wpositive, fatherId=fReference[0]}
  [1044] = {x=365.786, y=-228.104, rx=180, rz=-162.262, shoulder=lefty, elbow=epositive, wrist=wpositive, fatherId=fReference[0]}
  [1045] = {x=367.166, y=-228.546, rx=-180, rz=-162.424, shoulder=lefty, elbow=epositive, wrist=wpositive, fatherId=fReference[0]}
  [1046] = {x=368.546, y=-228.983, rx=-180, rz=-162.586, shoulder=lefty, elbow=epositive, wrist=wpositive, fatherId=fReference[0]}
  [1047] = {x=369.927, y=-229.416, rx=-180, rz=-162.75, shoulder=lefty, elbow=epositive, wrist=wpositive, fatherId=fReference[0]}
  [1048] = {x=371.309, y=-229.845, rx=-180, rz=-162.913, shoulder=lefty, elbow=epositive, wrist=wpositive, fatherId=fReference[0]}
  [1049] = {x=372.691, y=-230.27, rx=180, rz=-163.078, shoulder=lefty, elbow=epositive, wrist=wpositive, fatherId=fReference[0]}
  [1050] = {x=374.074, y=-230.69, rx=-180, rz=-163.243, shoulder=lefty, elbow=epositive, wrist=wpositive, fatherId=fReference[0]}
  [1051] = {x=375.457, y=-231.107, rx=-180, rz=-163.409, shoulder=lefty, elbow=epositive, wrist=wpositive, fatherId=fReference[0]}
  [1052] = {x=376.841, y=-231.519, rx=180, rz=-163.576, shoulder=lefty, elbow=epositive, wrist=wpositive, fatherId=fReference[0]}
  [1053] = {x=378.226, y=-231.928, rx=-180, rz=-163.743, shoulder=lefty, elbow=epositive, wrist=wpositive, fatherId=fReference[0]}
  [1054] = {x=379.611, y=-232.331, rx=-180, rz=-163.911, shoulder=lefty, elbow=epositive, wrist=wpositive, fatherId=fReference[0]}
  [1055] = {x=380.997, y=-232.731, rx=-180, rz=-164.08, shoulder=lefty, elbow=epositive, wrist=wpositive, fatherId=fReference[0]}
  [1056] = {x=382.384, y=-233.127, rx=180, rz=-164.249, shoulder=lefty, elbow=epositive, wrist=wpositive, fatherId=fReference[0]}
  [1057] = {x=383.771, y=-233.518, rx=-180, rz=-164.419, shoulder=lefty, elbow=epositive, wrist=wpositive, fatherId=fReference[0]}
  [1058] = {x=385.159, y=-233.905, rx=-180, rz=-164.589, shoulder=lefty, elbow=epositive, wrist=wpositive, fatherId=fReference[0]}
  [1059] = {x=386.547, y=-234.288, rx=180, rz=-164.76, shoulder=lefty, elbow=epositive, wrist=wpositive, fatherId=fReference[0]}
  [1060] = {x=387.936, y=-234.666, rx=180, rz=-164.932, shoulder=lefty, elbow=epositive, wrist=wpositive, fatherId=fReference[0]}
  [1061] = {x=389.325, y=-235.04, rx=180, rz=-165.105, shoulder=lefty, elbow=epositive, wrist=wpositive, fatherId=fReference[0]}
  [1062] = {x=390.715, y=-235.41, rx=180, rz=-165.277, shoulder=lefty, elbow=epositive, wrist=wpositive, fatherId=fReference[0]}
  [1063] = {x=392.106, y=-235.775, rx=-180, rz=-165.451, shoulder=lefty, elbow=epositive, wrist=wpositive, fatherId=fReference[0]}
  [1064] = {x=393.497, y=-236.136, rx=-180, rz=-165.625, shoulder=lefty, elbow=epositive, wrist=wpositive, fatherId=fReference[0]}
  [1065] = {x=394.889, y=-236.493, rx=180, rz=-165.8, shoulder=lefty, elbow=epositive, wrist=wpositive, fatherId=fReference[0]}
  [1066] = {x=396.281, y=-236.845, rx=-180, rz=-165.976, shoulder=lefty, elbow=epositive, wrist=wpositive, fatherId=fReference[0]}
  [1067] = {x=397.674, y=-237.193, rx=-180, rz=-166.152, shoulder=lefty, elbow=epositive, wrist=wpositive, fatherId=fReference[0]}
  [1068] = {x=399.068, y=-237.537, rx=-180, rz=-166.328, shoulder=lefty, elbow=epositive, wrist=wpositive, fatherId=fReference[0]}
  [1069] = {x=400.462, y=-237.876, rx=-180, rz=-166.505, shoulder=lefty, elbow=epositive, wrist=wpositive, fatherId=fReference[0]}
  [1070] = {x=401.856, y=-238.21, rx=-180, rz=-166.683, shoulder=lefty, elbow=epositive, wrist=wpositive, fatherId=fReference[0]}
  [1071] = {x=403.251, y=-238.541, rx=180, rz=-166.861, shoulder=lefty, elbow=epositive, wrist=wpositive, fatherId=fReference[0]}
  [1072] = {x=404.647, y=-238.866, rx=-180, rz=-167.04, shoulder=lefty, elbow=epositive, wrist=wpositive, fatherId=fReference[0]}
  [1073] = {x=406.043, y=-239.188, rx=-180, rz=-167.22, shoulder=lefty, elbow=epositive, wrist=wpositive, fatherId=fReference[0]}
  [1074] = {x=407.439, y=-239.505, rx=-180, rz=-167.4, shoulder=lefty, elbow=epositive, wrist=wpositive, fatherId=fReference[0]}
  [1075] = {x=408.836, y=-239.817, rx=180, rz=-167.581, shoulder=lefty, elbow=epositive, wrist=wpositive, fatherId=fReference[0]}
  [1076] = {x=410.234, y=-240.125, rx=180, rz=-167.762, shoulder=lefty, elbow=epositive, wrist=wpositive, fatherId=fReference[0]}
  [1077] = {x=411.632, y=-240.428, rx=-180, rz=-167.943, shoulder=lefty, elbow=epositive, wrist=wpositive, fatherId=fReference[0]}
  [1078] = {x=413.031, y=-240.727, rx=-180, rz=-168.126, shoulder=lefty, elbow=epositive, wrist=wpositive, fatherId=fReference[0]}
  [1079] = {x=414.43, y=-241.021, rx=180, rz=-168.308, shoulder=lefty, elbow=epositive, wrist=wpositive, fatherId=fReference[0]}
  [1080] = {x=415.829, y=-241.31, rx=180, rz=-168.492, shoulder=lefty, elbow=epositive, wrist=wpositive, fatherId=fReference[0]}
  [1081] = {x=417.229, y=-241.595, rx=180, rz=-168.675, shoulder=lefty, elbow=epositive, wrist=wpositive, fatherId=fReference[0]}
  [1082] = {x=418.63, y=-241.876, rx=-180, rz=-168.86, shoulder=lefty, elbow=epositive, wrist=wpositive, fatherId=fReference[0]}
  [1083] = {x=420.031, y=-242.152, rx=-180, rz=-169.045, shoulder=lefty, elbow=epositive, wrist=wpositive, fatherId=fReference[0]}
  [1084] = {x=421.432, y=-242.423, rx=-180, rz=-169.23, shoulder=lefty, elbow=epositive, wrist=wpositive, fatherId=fReference[0]}
  [1085] = {x=422.834, y=-242.69, rx=180, rz=-169.416, shoulder=lefty, elbow=epositive, wrist=wpositive, fatherId=fReference[0]}
  [1086] = {x=424.236, y=-242.952, rx=-180, rz=-169.602, shoulder=lefty, elbow=epositive, wrist=wpositive, fatherId=fReference[0]}
  [1087] = {x=425.639, y=-243.209, rx=-180, rz=-169.789, shoulder=lefty, elbow=epositive, wrist=wpositive, fatherId=fReference[0]}
  [1088] = {x=427.042, y=-243.462, rx=180, rz=-169.976, shoulder=lefty, elbow=epositive, wrist=wpositive, fatherId=fReference[0]}
  [1089] = {x=428.445, y=-243.71, rx=-180, rz=-170.164, shoulder=lefty, elbow=epositive, wrist=wpositive, fatherId=fReference[0]}
  [1090] = {x=429.849, y=-243.953, rx=180, rz=-170.352, shoulder=lefty, elbow=epositive, wrist=wpositive, fatherId=fReference[0]}
  [1091] = {x=431.254, y=-244.192, rx=180, rz=-170.54, shoulder=lefty, elbow=epositive, wrist=wpositive, fatherId=fReference[0]}
  [1092] = {x=432.658, y=-244.426, rx=-180, rz=-170.729, shoulder=lefty, elbow=epositive, wrist=wpositive, fatherId=fReference[0]}
  [1093] = {x=434.064, y=-244.655, rx=-180, rz=-170.919, shoulder=lefty, elbow=epositive, wrist=wpositive, fatherId=fReference[0]}
  [1094] = {x=435.469, y=-244.88, rx=-180, rz=-171.109, shoulder=lefty, elbow=epositive, wrist=wpositive, fatherId=fReference[0]}
  [1095] = {x=436.875, y=-245.1, rx=-180, rz=-171.299, shoulder=lefty, elbow=epositive, wrist=wpositive, fatherId=fReference[0]}
  [1096] = {x=438.281, y=-245.315, rx=180, rz=-171.49, shoulder=lefty, elbow=epositive, wrist=wpositive, fatherId=fReference[0]}
  [1097] = {x=439.688, y=-245.526, rx=180, rz=-171.681, shoulder=lefty, elbow=epositive, wrist=wpositive, fatherId=fReference[0]}
  [1098] = {x=441.095, y=-245.731, rx=-180, rz=-171.873, shoulder=lefty, elbow=epositive, wrist=wpositive, fatherId=fReference[0]}
  [1099] = {x=442.502, y=-245.932, rx=180, rz=-172.065, shoulder=lefty, elbow=epositive, wrist=wpositive, fatherId=fReference[0]}
  [1100] = {x=443.91, y=-246.129, rx=-180, rz=-172.257, shoulder=lefty, elbow=epositive, wrist=wpositive, fatherId=fReference[0]}
  [1101] = {x=445.318, y=-246.32, rx=180, rz=-172.449, shoulder=lefty, elbow=epositive, wrist=wpositive, fatherId=fReference[0]}
  [1102] = {x=446.726, y=-246.507, rx=180, rz=-172.643, shoulder=lefty, elbow=epositive, wrist=wpositive, fatherId=fReference[0]}
  [1103] = {x=448.134, y=-246.689, rx=-180, rz=-172.836, shoulder=lefty, elbow=epositive, wrist=wpositive, fatherId=fReference[0]}
  [1104] = {x=449.543, y=-246.866, rx=180, rz=-173.03, shoulder=lefty, elbow=epositive, wrist=wpositive, fatherId=fReference[0]}
  [1105] = {x=450.953, y=-247.038, rx=-180, rz=-173.224, shoulder=lefty, elbow=epositive, wrist=wpositive, fatherId=fReference[0]}
  [1106] = {x=452.362, y=-247.205, rx=-180, rz=-173.418, shoulder=lefty, elbow=epositive, wrist=wpositive, fatherId=fReference[0]}
  [1107] = {x=453.772, y=-247.368, rx=-180, rz=-173.613, shoulder=lefty, elbow=epositive, wrist=wpositive, fatherId=fReference[0]}
  [1108] = {x=455.182, y=-247.526, rx=180, rz=-173.808, shoulder=lefty, elbow=epositive, wrist=wpositive, fatherId=fReference[0]}
  [1109] = {x=456.592, y=-247.679, rx=180, rz=-174.003, shoulder=lefty, elbow=epositive, wrist=wpositive, fatherId=fReference[0]}
  [1110] = {x=458.003, y=-247.827, rx=-180, rz=-174.199, shoulder=lefty, elbow=epositive, wrist=wpositive, fatherId=fReference[0]}
  [1111] = {x=459.414, y=-247.971, rx=-180, rz=-174.395, shoulder=lefty, elbow=epositive, wrist=wpositive, fatherId=fReference[0]}
  [1112] = {x=460.825, y=-248.109, rx=180, rz=-174.591, shoulder=lefty, elbow=epositive, wrist=wpositive, fatherId=fReference[0]}
  [1113] = {x=462.236, y=-248.243, rx=-180, rz=-174.787, shoulder=lefty, elbow=epositive, wrist=wpositive, fatherId=fReference[0]}
  [1114] = {x=463.647, y=-248.371, rx=-180, rz=-174.984, shoulder=lefty, elbow=epositive, wrist=wpositive, fatherId=fReference[0]}
  [1115] = {x=465.059, y=-248.495, rx=180, rz=-175.181, shoulder=lefty, elbow=epositive, wrist=wpositive, fatherId=fReference[0]}
  [1116] = {x=466.471, y=-248.614, rx=180, rz=-175.378, shoulder=lefty, elbow=epositive, wrist=wpositive, fatherId=fReference[0]}
  [1117] = {x=467.883, y=-248.729, rx=-180, rz=-175.575, shoulder=lefty, elbow=epositive, wrist=wpositive, fatherId=fReference[0]}
  [1118] = {x=469.296, y=-248.838, rx=180, rz=-175.773, shoulder=lefty, elbow=epositive, wrist=wpositive, fatherId=fReference[0]}
  [1119] = {x=470.708, y=-248.942, rx=-180, rz=-175.971, shoulder=lefty, elbow=epositive, wrist=wpositive, fatherId=fReference[0]}
  [1120] = {x=472.121, y=-249.042, rx=-180, rz=-176.169, shoulder=lefty, elbow=epositive, wrist=wpositive, fatherId=fReference[0]}
  [1121] = {x=473.534, y=-249.136, rx=180, rz=-176.367, shoulder=lefty, elbow=epositive, wrist=wpositive, fatherId=fReference[0]}
  [1122] = {x=474.947, y=-249.226, rx=-180, rz=-176.566, shoulder=lefty, elbow=epositive, wrist=wpositive, fatherId=fReference[0]}
  [1123] = {x=476.36, y=-249.311, rx=-180, rz=-176.764, shoulder=lefty, elbow=epositive, wrist=wpositive, fatherId=fReference[0]}
  [1124] = {x=477.773, y=-249.391, rx=-180, rz=-176.963, shoulder=lefty, elbow=epositive, wrist=wpositive, fatherId=fReference[0]}
  [1125] = {x=479.187, y=-249.466, rx=-180, rz=-177.162, shoulder=lefty, elbow=epositive, wrist=wpositive, fatherId=fReference[0]}
  [1126] = {x=480.6, y=-249.536, rx=-180, rz=-177.361, shoulder=lefty, elbow=epositive, wrist=wpositive, fatherId=fReference[0]}
  [1127] = {x=482.014, y=-249.601, rx=180, rz=-177.56, shoulder=lefty, elbow=epositive, wrist=wpositive, fatherId=fReference[0]}
  [1128] = {x=483.428, y=-249.661, rx=-180, rz=-177.759, shoulder=lefty, elbow=epositive, wrist=wpositive, fatherId=fReference[0]}
  [1129] = {x=484.841, y=-249.717, rx=180, rz=-177.959, shoulder=lefty, elbow=epositive, wrist=wpositive, fatherId=fReference[0]}
  [1130] = {x=486.255, y=-249.767, rx=180, rz=-178.158, shoulder=lefty, elbow=epositive, wrist=wpositive, fatherId=fReference[0]}
  [1131] = {x=487.669, y=-249.812, rx=180, rz=-178.358, shoulder=lefty, elbow=epositive, wrist=wpositive, fatherId=fReference[0]}
  [1132] = {x=489.084, y=-249.853, rx=-180, rz=-178.557, shoulder=lefty, elbow=epositive, wrist=wpositive, fatherId=fReference[0]}
  [1133] = {x=490.498, y=-249.889, rx=-180, rz=-178.757, shoulder=lefty, elbow=epositive, wrist=wpositive, fatherId=fReference[0]}
  [1134] = {x=491.912, y=-249.919, rx=-180, rz=-178.957, shoulder=lefty, elbow=epositive, wrist=wpositive, fatherId=fReference[0]}
  [1135] = {x=493.326, y=-249.945, rx=180, rz=-179.157, shoulder=lefty, elbow=epositive, wrist=wpositive, fatherId=fReference[0]}
  [1136] = {x=494.741, y=-249.966, rx=180, rz=-179.357, shoulder=lefty, elbow=epositive, wrist=wpositive, fatherId=fReference[0]}
  [1137] = {x=496.155, y=-249.982, rx=-180, rz=-179.557, shoulder=lefty, elbow=epositive, wrist=wpositive, fatherId=fReference[0]}
  [1138] = {x=497.569, y=-249.993, rx=180, rz=-179.756, shoulder=lefty, elbow=epositive, wrist=wpositive, fatherId=fReference[0]}
  [1139] = {x=498.984, y=-249.999, rx=-180, rz=-179.956, shoulder=lefty, elbow=epositive, wrist=wpositive, fatherId=fReference[0]}
  [1140] = {x=500.398, y=-250, rx=-180, rz=179.844, shoulder=lefty, elbow=epositive, wrist=wpositive, fatherId=fReference[0]}
  [1141] = {x=501.812, y=-249.996, rx=-180, rz=179.644, shoulder=lefty, elbow=epositive, wrist=wpositive, fatherId=fReference[0]}
  [1142] = {x=503.227, y=-249.987, rx=180, rz=179.444, shoulder=lefty, elbow=epositive, wrist=wpositive, fatherId=fReference[0]}
  [1143] = {x=504.641, y=-249.973, rx=-180, rz=179.244, shoulder=lefty, elbow=epositive, wrist=wpositive, fatherId=fReference[0]}
  [1144] = {x=506.055, y=-249.955, rx=-180, rz=179.044, shoulder=lefty, elbow=epositive, wrist=wpositive, fatherId=fReference[0]}
  [1145] = {x=507.47, y=-249.931, rx=-180, rz=178.844, shoulder=lefty, elbow=epositive, wrist=wpositive, fatherId=fReference[0]}
  [1146] = {x=508.884, y=-249.903, rx=-180, rz=178.645, shoulder=lefty, elbow=epositive, wrist=wpositive, fatherId=fReference[0]}
  [1147] = {x=510.298, y=-249.869, rx=180, rz=178.445, shoulder=lefty, elbow=epositive, wrist=wpositive, fatherId=fReference[0]}
  [1148] = {x=511.712, y=-249.831, rx=180, rz=178.245, shoulder=lefty, elbow=epositive, wrist=wpositive, fatherId=fReference[0]}
  [1149] = {x=513.126, y=-249.787, rx=-180, rz=178.046, shoulder=lefty, elbow=epositive, wrist=wpositive, fatherId=fReference[0]}
  [1150] = {x=514.54, y=-249.739, rx=180, rz=177.846, shoulder=lefty, elbow=epositive, wrist=wpositive, fatherId=fReference[0]}
  [1151] = {x=515.954, y=-249.686, rx=180, rz=177.647, shoulder=lefty, elbow=epositive, wrist=wpositive, fatherId=fReference[0]}
  [1152] = {x=517.368, y=-249.628, rx=-180, rz=177.448, shoulder=lefty, elbow=epositive, wrist=wpositive, fatherId=fReference[0]}
  [1153] = {x=518.782, y=-249.565, rx=-180, rz=177.249, shoulder=lefty, elbow=epositive, wrist=wpositive, fatherId=fReference[0]}
  [1154] = {x=520.195, y=-249.497, rx=-180, rz=177.05, shoulder=lefty, elbow=epositive, wrist=wpositive, fatherId=fReference[0]}
  [1155] = {x=521.609, y=-249.424, rx=180, rz=176.851, shoulder=lefty, elbow=epositive, wrist=wpositive, fatherId=fReference[0]}
  [1156] = {x=523.022, y=-249.346, rx=-180, rz=176.652, shoulder=lefty, elbow=epositive, wrist=wpositive, fatherId=fReference[0]}
  [1157] = {x=524.435, y=-249.264, rx=-180, rz=176.454, shoulder=lefty, elbow=epositive, wrist=wpositive, fatherId=fReference[0]}
  [1158] = {x=525.848, y=-249.176, rx=180, rz=176.256, shoulder=lefty, elbow=epositive, wrist=wpositive, fatherId=fReference[0]}
  [1159] = {x=527.261, y=-249.084, rx=-180, rz=176.058, shoulder=lefty, elbow=epositive, wrist=wpositive, fatherId=fReference[0]}
  [1160] = {x=528.674, y=-248.986, rx=-180, rz=175.86, shoulder=lefty, elbow=epositive, wrist=wpositive, fatherId=fReference[0]}
  [1161] = {x=530.086, y=-248.884, rx=-180, rz=175.662, shoulder=lefty, elbow=epositive, wrist=wpositive, fatherId=fReference[0]}
  [1162] = {x=531.498, y=-248.777, rx=-180, rz=175.465, shoulder=lefty, elbow=epositive, wrist=wpositive, fatherId=fReference[0]}
  [1163] = {x=532.911, y=-248.665, rx=-180, rz=175.267, shoulder=lefty, elbow=epositive, wrist=wpositive, fatherId=fReference[0]}
  [1164] = {x=534.323, y=-248.548, rx=180, rz=175.07, shoulder=lefty, elbow=epositive, wrist=wpositive, fatherId=fReference[0]}
  [1165] = {x=535.734, y=-248.426, rx=180, rz=174.874, shoulder=lefty, elbow=epositive, wrist=wpositive, fatherId=fReference[0]}
  [1166] = {x=537.146, y=-248.3, rx=180, rz=174.677, shoulder=lefty, elbow=epositive, wrist=wpositive, fatherId=fReference[0]}
  [1167] = {x=538.557, y=-248.168, rx=-180, rz=174.481, shoulder=lefty, elbow=epositive, wrist=wpositive, fatherId=fReference[0]}
  [1168] = {x=539.968, y=-248.032, rx=-180, rz=174.285, shoulder=lefty, elbow=epositive, wrist=wpositive, fatherId=fReference[0]}
  [1169] = {x=541.379, y=-247.891, rx=180, rz=174.089, shoulder=lefty, elbow=epositive, wrist=wpositive, fatherId=fReference[0]}
  [1170] = {x=542.79, y=-247.744, rx=-180, rz=173.894, shoulder=lefty, elbow=epositive, wrist=wpositive, fatherId=fReference[0]}
  [1171] = {x=544.2, y=-247.594, rx=-180, rz=173.698, shoulder=lefty, elbow=epositive, wrist=wpositive, fatherId=fReference[0]}
  [1172] = {x=545.61, y=-247.438, rx=-180, rz=173.504, shoulder=lefty, elbow=epositive, wrist=wpositive, fatherId=fReference[0]}
  [1173] = {x=547.02, y=-247.277, rx=180, rz=173.309, shoulder=lefty, elbow=epositive, wrist=wpositive, fatherId=fReference[0]}
  [1174] = {x=548.43, y=-247.112, rx=180, rz=173.115, shoulder=lefty, elbow=epositive, wrist=wpositive, fatherId=fReference[0]}
  [1175] = {x=549.839, y=-246.942, rx=-180, rz=172.921, shoulder=lefty, elbow=epositive, wrist=wpositive, fatherId=fReference[0]}
  [1176] = {x=551.248, y=-246.767, rx=-180, rz=172.727, shoulder=lefty, elbow=epositive, wrist=wpositive, fatherId=fReference[0]}
  [1177] = {x=552.657, y=-246.587, rx=-180, rz=172.534, shoulder=lefty, elbow=epositive, wrist=wpositive, fatherId=fReference[0]}
  [1178] = {x=554.065, y=-246.402, rx=-180, rz=172.341, shoulder=lefty, elbow=epositive, wrist=wpositive, fatherId=fReference[0]}
  [1179] = {x=555.473, y=-246.213, rx=180, rz=172.149, shoulder=lefty, elbow=epositive, wrist=wpositive, fatherId=fReference[0]}
  [1180] = {x=556.881, y=-246.019, rx=-180, rz=171.957, shoulder=lefty, elbow=epositive, wrist=wpositive, fatherId=fReference[0]}
  [1181] = {x=558.289, y=-245.82, rx=-180, rz=171.765, shoulder=lefty, elbow=epositive, wrist=wpositive, fatherId=fReference[0]}
  [1182] = {x=559.696, y=-245.616, rx=-180, rz=171.574, shoulder=lefty, elbow=epositive, wrist=wpositive, fatherId=fReference[0]}
  [1183] = {x=561.102, y=-245.408, rx=-180, rz=171.383, shoulder=lefty, elbow=epositive, wrist=wpositive, fatherId=fReference[0]}
  [1184] = {x=562.509, y=-245.195, rx=-180, rz=171.192, shoulder=lefty, elbow=epositive, wrist=wpositive, fatherId=fReference[0]}
  [1185] = {x=563.915, y=-244.977, rx=-180, rz=171.002, shoulder=lefty, elbow=epositive, wrist=wpositive, fatherId=fReference[0]}
  [1186] = {x=565.321, y=-244.755, rx=-180, rz=170.813, shoulder=lefty, elbow=epositive, wrist=wpositive, fatherId=fReference[0]}
  [1187] = {x=566.726, y=-244.527, rx=-180, rz=170.623, shoulder=lefty, elbow=epositive, wrist=wpositive, fatherId=fReference[0]}
  [1188] = {x=568.131, y=-244.295, rx=180, rz=170.435, shoulder=lefty, elbow=epositive, wrist=wpositive, fatherId=fReference[0]}
  [1189] = {x=569.535, y=-244.059, rx=-180, rz=170.246, shoulder=lefty, elbow=epositive, wrist=wpositive, fatherId=fReference[0]}
  [1190] = {x=570.939, y=-243.817, rx=180, rz=170.058, shoulder=lefty, elbow=epositive, wrist=wpositive, fatherId=fReference[0]}
  [1191] = {x=572.343, y=-243.571, rx=180, rz=169.871, shoulder=lefty, elbow=epositive, wrist=wpositive, fatherId=fReference[0]}
  [1192] = {x=573.746, y=-243.32, rx=-180, rz=169.684, shoulder=lefty, elbow=epositive, wrist=wpositive, fatherId=fReference[0]}
  [1193] = {x=575.149, y=-243.065, rx=-180, rz=169.497, shoulder=lefty, elbow=epositive, wrist=wpositive, fatherId=fReference[0]}
  [1194] = {x=576.552, y=-242.805, rx=-180, rz=169.311, shoulder=lefty, elbow=epositive, wrist=wpositive, fatherId=fReference[0]}
  [1195] = {x=577.954, y=-242.54, rx=-180, rz=169.126, shoulder=lefty, elbow=epositive, wrist=wpositive, fatherId=fReference[0]}
  [1196] = {x=579.355, y=-242.271, rx=180, rz=168.941, shoulder=lefty, elbow=epositive, wrist=wpositive, fatherId=fReference[0]}
  [1197] = {x=580.757, y=-241.997, rx=180, rz=168.756, shoulder=lefty, elbow=epositive, wrist=wpositive, fatherId=fReference[0]}
  [1198] = {x=582.157, y=-241.719, rx=-180, rz=168.572, shoulder=lefty, elbow=epositive, wrist=wpositive, fatherId=fReference[0]}
  [1199] = {x=583.557, y=-241.436, rx=-180, rz=168.389, shoulder=lefty, elbow=epositive, wrist=wpositive, fatherId=fReference[0]}
  [1200] = {x=584.957, y=-241.148, rx=180, rz=168.206, shoulder=lefty, elbow=epositive, wrist=wpositive, fatherId=fReference[0]}
  [1201] = {x=586.357, y=-240.856, rx=-180, rz=168.023, shoulder=lefty, elbow=epositive, wrist=wpositive, fatherId=fReference[0]}
  [1202] = {x=587.755, y=-240.559, rx=180, rz=167.841, shoulder=lefty, elbow=epositive, wrist=wpositive, fatherId=fReference[0]}
  [1203] = {x=589.154, y=-240.258, rx=-180, rz=167.66, shoulder=lefty, elbow=epositive, wrist=wpositive, fatherId=fReference[0]}
  [1204] = {x=590.552, y=-239.952, rx=-180, rz=167.479, shoulder=lefty, elbow=epositive, wrist=wpositive, fatherId=fReference[0]}
  [1205] = {x=591.949, y=-239.642, rx=180, rz=167.299, shoulder=lefty, elbow=epositive, wrist=wpositive, fatherId=fReference[0]}
  [1206] = {x=593.346, y=-239.327, rx=180, rz=167.119, shoulder=lefty, elbow=epositive, wrist=wpositive, fatherId=fReference[0]}
  [1207] = {x=594.742, y=-239.008, rx=-180, rz=166.94, shoulder=lefty, elbow=epositive, wrist=wpositive, fatherId=fReference[0]}
  [1208] = {x=596.138, y=-238.684, rx=180, rz=166.761, shoulder=lefty, elbow=epositive, wrist=wpositive, fatherId=fReference[0]}
  [1209] = {x=597.533, y=-238.356, rx=180, rz=166.583, shoulder=lefty, elbow=epositive, wrist=wpositive, fatherId=fReference[0]}
  [1210] = {x=598.928, y=-238.023, rx=-180, rz=166.405, shoulder=lefty, elbow=epositive, wrist=wpositive, fatherId=fReference[0]}
  [1211] = {x=600.322, y=-237.686, rx=180, rz=166.229, shoulder=lefty, elbow=epositive, wrist=wpositive, fatherId=fReference[0]}
  [1212] = {x=601.716, y=-237.344, rx=180, rz=166.052, shoulder=lefty, elbow=epositive, wrist=wpositive, fatherId=fReference[0]}
  [1213] = {x=603.109, y=-236.998, rx=180, rz=165.877, shoulder=lefty, elbow=epositive, wrist=wpositive, fatherId=fReference[0]}
  [1214] = {x=604.502, y=-236.648, rx=-180, rz=165.702, shoulder=lefty, elbow=epositive, wrist=wpositive, fatherId=fReference[0]}
  [1215] = {x=605.894, y=-236.293, rx=-180, rz=165.527, shoulder=lefty, elbow=epositive, wrist=wpositive, fatherId=fReference[0]}
  [1216] = {x=607.286, y=-235.934, rx=-180, rz=165.353, shoulder=lefty, elbow=epositive, wrist=wpositive, fatherId=fReference[0]}
  [1217] = {x=608.677, y=-235.57, rx=180, rz=165.18, shoulder=lefty, elbow=epositive, wrist=wpositive, fatherId=fReference[0]}
  [1218] = {x=610.067, y=-235.202, rx=-180, rz=165.007, shoulder=lefty, elbow=epositive, wrist=wpositive, fatherId=fReference[0]}
  [1219] = {x=611.457, y=-234.83, rx=-180, rz=164.835, shoulder=lefty, elbow=epositive, wrist=wpositive, fatherId=fReference[0]}
  [1220] = {x=612.846, y=-234.454, rx=180, rz=164.664, shoulder=lefty, elbow=epositive, wrist=wpositive, fatherId=fReference[0]}
  [1221] = {x=614.235, y=-234.073, rx=-180, rz=164.493, shoulder=lefty, elbow=epositive, wrist=wpositive, fatherId=fReference[0]}
  [1222] = {x=615.623, y=-233.688, rx=-180, rz=164.323, shoulder=lefty, elbow=epositive, wrist=wpositive, fatherId=fReference[0]}
  [1223] = {x=617.01, y=-233.298, rx=180, rz=164.153, shoulder=lefty, elbow=epositive, wrist=wpositive, fatherId=fReference[0]}
  [1224] = {x=618.397, y=-232.905, rx=-180, rz=163.985, shoulder=lefty, elbow=epositive, wrist=wpositive, fatherId=fReference[0]}
  [1225] = {x=619.783, y=-232.507, rx=180, rz=163.816, shoulder=lefty, elbow=epositive, wrist=wpositive, fatherId=fReference[0]}
  [1226] = {x=621.169, y=-232.104, rx=180, rz=163.649, shoulder=lefty, elbow=epositive, wrist=wpositive, fatherId=fReference[0]}
  [1227] = {x=622.554, y=-231.698, rx=-180, rz=163.482, shoulder=lefty, elbow=epositive, wrist=wpositive, fatherId=fReference[0]}
  [1228] = {x=623.939, y=-231.288, rx=180, rz=163.316, shoulder=lefty, elbow=epositive, wrist=wpositive, fatherId=fReference[0]}
  [1229] = {x=625.322, y=-230.873, rx=-180, rz=163.15, shoulder=lefty, elbow=epositive, wrist=wpositive, fatherId=fReference[0]}
  [1230] = {x=626.706, y=-230.454, rx=180, rz=162.985, shoulder=lefty, elbow=epositive, wrist=wpositive, fatherId=fReference[0]}
  [1231] = {x=628.088, y=-230.031, rx=180, rz=162.821, shoulder=lefty, elbow=epositive, wrist=wpositive, fatherId=fReference[0]}
  [1232] = {x=629.47, y=-229.604, rx=-180, rz=162.657, shoulder=lefty, elbow=epositive, wrist=wpositive, fatherId=fReference[0]}
  [1233] = {x=630.851, y=-229.172, rx=-180, rz=162.494, shoulder=lefty, elbow=epositive, wrist=wpositive, fatherId=fReference[0]}
  [1234] = {x=632.232, y=-228.737, rx=180, rz=162.332, shoulder=lefty, elbow=epositive, wrist=wpositive, fatherId=fReference[0]}
  [1235] = {x=633.612, y=-228.297, rx=-180, rz=162.171, shoulder=lefty, elbow=epositive, wrist=wpositive, fatherId=fReference[0]}
  [1236] = {x=634.991, y=-227.854, rx=-180, rz=162.01, shoulder=lefty, elbow=epositive, wrist=wpositive, fatherId=fReference[0]}
  [1237] = {x=636.37, y=-227.406, rx=-180, rz=161.85, shoulder=lefty, elbow=epositive, wrist=wpositive, fatherId=fReference[0]}
  [1238] = {x=637.748, y=-226.954, rx=-180, rz=161.69, shoulder=lefty, elbow=epositive, wrist=wpositive, fatherId=fReference[0]}
  [1239] = {x=639.125, y=-226.498, rx=-180, rz=161.531, shoulder=lefty, elbow=epositive, wrist=wpositive, fatherId=fReference[0]}
  [1240] = {x=640.502, y=-226.038, rx=180, rz=161.373, shoulder=lefty, elbow=epositive, wrist=wpositive, fatherId=fReference[0]}
  [1241] = {x=641.878, y=-225.575, rx=180, rz=161.216, shoulder=lefty, elbow=epositive, wrist=wpositive, fatherId=fReference[0]}
  [1242] = {x=643.254, y=-225.107, rx=180, rz=161.059, shoulder=lefty, elbow=epositive, wrist=wpositive, fatherId=fReference[0]}
  [1243] = {x=644.628, y=-224.635, rx=180, rz=160.903, shoulder=lefty, elbow=epositive, wrist=wpositive, fatherId=fReference[0]}
  [1244] = {x=646.002, y=-224.159, rx=180, rz=160.748, shoulder=lefty, elbow=epositive, wrist=wpositive, fatherId=fReference[0]}
  [1245] = {x=647.376, y=-223.68, rx=180, rz=160.593, shoulder=lefty, elbow=epositive, wrist=wpositive, fatherId=fReference[0]}
  [1246] = {x=648.748, y=-223.196, rx=180, rz=160.439, shoulder=lefty, elbow=epositive, wrist=wpositive, fatherId=fReference[0]}
  [1247] = {x=650.12, y=-222.709, rx=-180, rz=160.286, shoulder=lefty, elbow=epositive, wrist=wpositive, fatherId=fReference[0]}
  [1248] = {x=651.491, y=-222.217, rx=-180, rz=160.133, shoulder=lefty, elbow=epositive, wrist=wpositive, fatherId=fReference[0]}
  [1249] = {x=652.862, y=-221.722, rx=180, rz=159.981, shoulder=lefty, elbow=epositive, wrist=wpositive, fatherId=fReference[0]}
  [1250] = {x=654.232, y=-221.223, rx=180, rz=159.83, shoulder=lefty, elbow=epositive, wrist=wpositive, fatherId=fReference[0]}
  [1251] = {x=655.601, y=-220.72, rx=-180, rz=159.68, shoulder=lefty, elbow=epositive, wrist=wpositive, fatherId=fReference[0]}
  [1252] = {x=656.969, y=-220.213, rx=180, rz=159.53, shoulder=lefty, elbow=epositive, wrist=wpositive, fatherId=fReference[0]}
  [1253] = {x=658.337, y=-219.703, rx=180, rz=159.381, shoulder=lefty, elbow=epositive, wrist=wpositive, fatherId=fReference[0]}
  [1254] = {x=659.704, y=-219.189, rx=-180, rz=159.233, shoulder=lefty, elbow=epositive, wrist=wpositive, fatherId=fReference[0]}
  [1255] = {x=661.07, y=-218.67, rx=180, rz=159.086, shoulder=lefty, elbow=epositive, wrist=wpositive, fatherId=fReference[0]}
  [1256] = {x=662.436, y=-218.149, rx=-180, rz=158.939, shoulder=lefty, elbow=epositive, wrist=wpositive, fatherId=fReference[0]}
  [1257] = {x=663.801, y=-217.623, rx=-180, rz=158.793, shoulder=lefty, elbow=epositive, wrist=wpositive, fatherId=fReference[0]}
  [1258] = {x=665.165, y=-217.094, rx=180, rz=158.647, shoulder=lefty, elbow=epositive, wrist=wpositive, fatherId=fReference[0]}
  [1259] = {x=666.528, y=-216.561, rx=180, rz=158.503, shoulder=lefty, elbow=epositive, wrist=wpositive, fatherId=fReference[0]}
  [1260] = {x=667.891, y=-216.024, rx=-180, rz=158.359, shoulder=lefty, elbow=epositive, wrist=wpositive, fatherId=fReference[0]}
  [1261] = {x=669.253, y=-215.484, rx=180, rz=158.216, shoulder=lefty, elbow=epositive, wrist=wpositive, fatherId=fReference[0]}
  [1262] = {x=670.614, y=-214.94, rx=180, rz=158.073, shoulder=lefty, elbow=epositive, wrist=wpositive, fatherId=fReference[0]}
  [1263] = {x=671.974, y=-214.392, rx=-180, rz=157.931, shoulder=lefty, elbow=epositive, wrist=wpositive, fatherId=fReference[0]}
  [1264] = {x=673.334, y=-213.841, rx=180, rz=157.79, shoulder=lefty, elbow=epositive, wrist=wpositive, fatherId=fReference[0]}
  [1265] = {x=674.693, y=-213.286, rx=180, rz=157.65, shoulder=lefty, elbow=epositive, wrist=wpositive, fatherId=fReference[0]}
  [1266] = {x=676.052, y=-212.727, rx=-180, rz=157.51, shoulder=lefty, elbow=epositive, wrist=wpositive, fatherId=fReference[0]}
  [1267] = {x=677.409, y=-212.165, rx=180, rz=157.371, shoulder=lefty, elbow=epositive, wrist=wpositive, fatherId=fReference[0]}
  [1268] = {x=678.766, y=-211.6, rx=180, rz=157.233, shoulder=lefty, elbow=epositive, wrist=wpositive, fatherId=fReference[0]}
  [1269] = {x=680.122, y=-211.031, rx=180, rz=157.096, shoulder=lefty, elbow=epositive, wrist=wpositive, fatherId=fReference[0]}
  [1270] = {x=681.477, y=-210.458, rx=-180, rz=156.959, shoulder=lefty, elbow=epositive, wrist=wpositive, fatherId=fReference[0]}
  [1271] = {x=682.832, y=-209.882, rx=180, rz=156.823, shoulder=lefty, elbow=epositive, wrist=wpositive, fatherId=fReference[0]}
  [1272] = {x=684.186, y=-209.302, rx=180, rz=156.688, shoulder=lefty, elbow=epositive, wrist=wpositive, fatherId=fReference[0]}
  [1273] = {x=685.539, y=-208.719, rx=-180, rz=156.553, shoulder=lefty, elbow=epositive, wrist=wpositive, fatherId=fReference[0]}
  [1274] = {x=686.891, y=-208.133, rx=180, rz=156.42, shoulder=lefty, elbow=epositive, wrist=wpositive, fatherId=fReference[0]}
  [1275] = {x=688.243, y=-207.543, rx=180, rz=156.287, shoulder=lefty, elbow=epositive, wrist=wpositive, fatherId=fReference[0]}
  [1276] = {x=689.593, y=-206.949, rx=180, rz=156.154, shoulder=lefty, elbow=epositive, wrist=wpositive, fatherId=fReference[0]}
  [1277] = {x=690.943, y=-206.353, rx=180, rz=156.023, shoulder=lefty, elbow=epositive, wrist=wpositive, fatherId=fReference[0]}
  [1278] = {x=692.293, y=-205.753, rx=180, rz=155.892, shoulder=lefty, elbow=epositive, wrist=wpositive, fatherId=fReference[0]}
  [1279] = {x=693.641, y=-205.149, rx=-180, rz=155.762, shoulder=lefty, elbow=epositive, wrist=wpositive, fatherId=fReference[0]}
  [1280] = {x=694.989, y=-204.542, rx=-180, rz=155.632, shoulder=lefty, elbow=epositive, wrist=wpositive, fatherId=fReference[0]}
  [1281] = {x=696.336, y=-203.932, rx=180, rz=155.503, shoulder=lefty, elbow=epositive, wrist=wpositive, fatherId=fReference[0]}
  [1282] = {x=697.682, y=-203.319, rx=-180, rz=155.375, shoulder=lefty, elbow=epositive, wrist=wpositive, fatherId=fReference[0]}
  [1283] = {x=699.028, y=-202.702, rx=-180, rz=155.248, shoulder=lefty, elbow=epositive, wrist=wpositive, fatherId=fReference[0]}
  [1284] = {x=700.373, y=-202.082, rx=180, rz=155.122, shoulder=lefty, elbow=epositive, wrist=wpositive, fatherId=fReference[0]}
  [1285] = {x=701.717, y=-201.459, rx=180, rz=154.996, shoulder=lefty, elbow=epositive, wrist=wpositive, fatherId=fReference[0]}
  [1286] = {x=703.06, y=-200.832, rx=180, rz=154.871, shoulder=lefty, elbow=epositive, wrist=wpositive, fatherId=fReference[0]}
  [1287] = {x=704.403, y=-200.203, rx=-180, rz=154.746, shoulder=lefty, elbow=epositive, wrist=wpositive, fatherId=fReference[0]}
  [1288] = {x=705.744, y=-199.57, rx=-180, rz=154.622, shoulder=lefty, elbow=epositive, wrist=wpositive, fatherId=fReference[0]}
  [1289] = {x=707.085, y=-198.933, rx=180, rz=154.499, shoulder=lefty, elbow=epositive, wrist=wpositive, fatherId=fReference[0]}
  [1290] = {x=708.426, y=-198.294, rx=-180, rz=154.377, shoulder=lefty, elbow=epositive, wrist=wpositive, fatherId=fReference[0]}
  [1291] = {x=709.765, y=-197.652, rx=180, rz=154.256, shoulder=lefty, elbow=epositive, wrist=wpositive, fatherId=fReference[0]}
  [1292] = {x=711.104, y=-197.006, rx=180, rz=154.135, shoulder=lefty, elbow=epositive, wrist=wpositive, fatherId=fReference[0]}
  [1293] = {x=712.442, y=-196.357, rx=-180, rz=154.015, shoulder=lefty, elbow=epositive, wrist=wpositive, fatherId=fReference[0]}
  [1294] = {x=713.779, y=-195.706, rx=180, rz=153.895, shoulder=lefty, elbow=epositive, wrist=wpositive, fatherId=fReference[0]}
  [1295] = {x=715.116, y=-195.051, rx=180, rz=153.776, shoulder=lefty, elbow=epositive, wrist=wpositive, fatherId=fReference[0]}
  [1296] = {x=716.452, y=-194.393, rx=-180, rz=153.658, shoulder=lefty, elbow=epositive, wrist=wpositive, fatherId=fReference[0]}
  [1297] = {x=717.787, y=-193.732, rx=180, rz=153.541, shoulder=lefty, elbow=epositive, wrist=wpositive, fatherId=fReference[0]}
  [1298] = {x=719.121, y=-193.067, rx=-180, rz=153.424, shoulder=lefty, elbow=epositive, wrist=wpositive, fatherId=fReference[0]}
  [1299] = {x=720.455, y=-192.4, rx=180, rz=153.309, shoulder=lefty, elbow=epositive, wrist=wpositive, fatherId=fReference[0]}
  [1300] = {x=721.788, y=-191.73, rx=180, rz=153.193, shoulder=lefty, elbow=epositive, wrist=wpositive, fatherId=fReference[0]}
  [1301] = {x=723.12, y=-191.057, rx=180, rz=153.079, shoulder=lefty, elbow=epositive, wrist=wpositive, fatherId=fReference[0]}
  [1302] = {x=724.451, y=-190.381, rx=180, rz=152.965, shoulder=lefty, elbow=epositive, wrist=wpositive, fatherId=fReference[0]}
  [1303] = {x=725.782, y=-189.702, rx=180, rz=152.852, shoulder=lefty, elbow=epositive, wrist=wpositive, fatherId=fReference[0]}
  [1304] = {x=727.112, y=-189.02, rx=-180, rz=152.739, shoulder=lefty, elbow=epositive, wrist=wpositive, fatherId=fReference[0]}
  [1305] = {x=728.441, y=-188.335, rx=-180, rz=152.628, shoulder=lefty, elbow=epositive, wrist=wpositive, fatherId=fReference[0]}
  [1306] = {x=729.77, y=-187.647, rx=180, rz=152.517, shoulder=lefty, elbow=epositive, wrist=wpositive, fatherId=fReference[0]}
  [1307] = {x=731.098, y=-186.957, rx=-180, rz=152.406, shoulder=lefty, elbow=epositive, wrist=wpositive, fatherId=fReference[0]}
  [1308] = {x=732.425, y=-186.263, rx=180, rz=152.297, shoulder=lefty, elbow=epositive, wrist=wpositive, fatherId=fReference[0]}
  [1309] = {x=733.751, y=-185.567, rx=180, rz=152.188, shoulder=lefty, elbow=epositive, wrist=wpositive, fatherId=fReference[0]}
  [1310] = {x=735.077, y=-184.867, rx=-180, rz=152.079, shoulder=lefty, elbow=epositive, wrist=wpositive, fatherId=fReference[0]}
  [1311] = {x=736.401, y=-184.165, rx=180, rz=151.972, shoulder=lefty, elbow=epositive, wrist=wpositive, fatherId=fReference[0]}
  [1312] = {x=737.726, y=-183.46, rx=-180, rz=151.865, shoulder=lefty, elbow=epositive, wrist=wpositive, fatherId=fReference[0]}
  [1313] = {x=739.049, y=-182.753, rx=-180, rz=151.759, shoulder=lefty, elbow=epositive, wrist=wpositive, fatherId=fReference[0]}
  [1314] = {x=740.372, y=-182.042, rx=180, rz=151.653, shoulder=lefty, elbow=epositive, wrist=wpositive, fatherId=fReference[0]}
  [1315] = {x=741.694, y=-181.329, rx=-180, rz=151.548, shoulder=lefty, elbow=epositive, wrist=wpositive, fatherId=fReference[0]}
  [1316] = {x=743.015, y=-180.613, rx=180, rz=151.444, shoulder=lefty, elbow=epositive, wrist=wpositive, fatherId=fReference[0]}
  [1317] = {x=744.336, y=-179.894, rx=180, rz=151.341, shoulder=lefty, elbow=epositive, wrist=wpositive, fatherId=fReference[0]}
  [1318] = {x=745.656, y=-179.173, rx=-180, rz=151.238, shoulder=lefty, elbow=epositive, wrist=wpositive, fatherId=fReference[0]}
  [1319] = {x=746.975, y=-178.449, rx=180, rz=151.136, shoulder=lefty, elbow=epositive, wrist=wpositive, fatherId=fReference[0]}
  [1320] = {x=748.293, y=-177.722, rx=180, rz=151.034, shoulder=lefty, elbow=epositive, wrist=wpositive, fatherId=fReference[0]}
  [1321] = {x=749.611, y=-176.993, rx=-180, rz=150.933, shoulder=lefty, elbow=epositive, wrist=wpositive, fatherId=fReference[0]}
  [1322] = {x=750.928, y=-176.26, rx=180, rz=150.833, shoulder=lefty, elbow=epositive, wrist=wpositive, fatherId=fReference[0]}
  [1323] = {x=752.244, y=-175.526, rx=180, rz=150.734, shoulder=lefty, elbow=epositive, wrist=wpositive, fatherId=fReference[0]}
  [1324] = {x=753.56, y=-174.788, rx=-180, rz=150.635, shoulder=lefty, elbow=epositive, wrist=wpositive, fatherId=fReference[0]}
  [1325] = {x=754.875, y=-174.049, rx=180, rz=150.537, shoulder=lefty, elbow=epositive, wrist=wpositive, fatherId=fReference[0]}
  [1326] = {x=756.189, y=-173.306, rx=180, rz=150.439, shoulder=lefty, elbow=epositive, wrist=wpositive, fatherId=fReference[0]}
  [1327] = {x=757.503, y=-172.561, rx=180, rz=150.342, shoulder=lefty, elbow=epositive, wrist=wpositive, fatherId=fReference[0]}
  [1328] = {x=758.816, y=-171.814, rx=180, rz=150.246, shoulder=lefty, elbow=epositive, wrist=wpositive, fatherId=fReference[0]}
  [1329] = {x=760.128, y=-171.064, rx=180, rz=150.151, shoulder=lefty, elbow=epositive, wrist=wpositive, fatherId=fReference[0]}
  [1330] = {x=761.439, y=-170.311, rx=180, rz=150.056, shoulder=lefty, elbow=epositive, wrist=wpositive, fatherId=fReference[0]}
  [1331] = {x=762.75, y=-169.556, rx=180, rz=149.961, shoulder=lefty, elbow=epositive, wrist=wpositive, fatherId=fReference[0]}
  [1332] = {x=764.06, y=-168.798, rx=180, rz=149.868, shoulder=lefty, elbow=epositive, wrist=wpositive, fatherId=fReference[0]}
  [1333] = {x=765.369, y=-168.038, rx=180, rz=149.775, shoulder=lefty, elbow=epositive, wrist=wpositive, fatherId=fReference[0]}
  [1334] = {x=766.678, y=-167.276, rx=-180, rz=149.683, shoulder=lefty, elbow=epositive, wrist=wpositive, fatherId=fReference[0]}
  [1335] = {x=767.986, y=-166.511, rx=180, rz=149.591, shoulder=lefty, elbow=epositive, wrist=wpositive, fatherId=fReference[0]}
  [1336] = {x=769.293, y=-165.744, rx=180, rz=149.5, shoulder=lefty, elbow=epositive, wrist=wpositive, fatherId=fReference[0]}
  [1337] = {x=770.6, y=-164.974, rx=-180, rz=149.41, shoulder=lefty, elbow=epositive, wrist=wpositive, fatherId=fReference[0]}
  [1338] = {x=771.906, y=-164.202, rx=180, rz=149.32, shoulder=lefty, elbow=epositive, wrist=wpositive, fatherId=fReference[0]}
  [1339] = {x=773.211, y=-163.428, rx=-180, rz=149.231, shoulder=lefty, elbow=epositive, wrist=wpositive, fatherId=fReference[0]}
  [1340] = {x=774.516, y=-162.651, rx=180, rz=149.142, shoulder=lefty, elbow=epositive, wrist=wpositive, fatherId=fReference[0]}
  [1341] = {x=775.82, y=-161.872, rx=180, rz=149.054, shoulder=lefty, elbow=epositive, wrist=wpositive, fatherId=fReference[0]}
  [1342] = {x=777.123, y=-161.091, rx=180, rz=148.967, shoulder=lefty, elbow=epositive, wrist=wpositive, fatherId=fReference[0]}
  [1343] = {x=778.425, y=-160.307, rx=180, rz=148.881, shoulder=lefty, elbow=epositive, wrist=wpositive, fatherId=fReference[0]}
  [1344] = {x=779.727, y=-159.521, rx=180, rz=148.795, shoulder=lefty, elbow=epositive, wrist=wpositive, fatherId=fReference[0]}
  [1345] = {x=781.028, y=-158.733, rx=-180, rz=148.709, shoulder=lefty, elbow=epositive, wrist=wpositive, fatherId=fReference[0]}
  [1346] = {x=782.329, y=-157.942, rx=-180, rz=148.625, shoulder=lefty, elbow=epositive, wrist=wpositive, fatherId=fReference[0]}
  [1347] = {x=783.629, y=-157.15, rx=-180, rz=148.54, shoulder=lefty, elbow=epositive, wrist=wpositive, fatherId=fReference[0]}
  [1348] = {x=784.928, y=-156.355, rx=180, rz=148.457, shoulder=lefty, elbow=epositive, wrist=wpositive, fatherId=fReference[0]}
  [1349] = {x=786.227, y=-155.558, rx=180, rz=148.374, shoulder=lefty, elbow=epositive, wrist=wpositive, fatherId=fReference[0]}
  [1350] = {x=787.524, y=-154.758, rx=180, rz=148.292, shoulder=lefty, elbow=epositive, wrist=wpositive, fatherId=fReference[0]}
  [1351] = {x=788.822, y=-153.957, rx=180, rz=148.21, shoulder=lefty, elbow=epositive, wrist=wpositive, fatherId=fReference[0]}
  [1352] = {x=790.118, y=-153.153, rx=-180, rz=148.129, shoulder=lefty, elbow=epositive, wrist=wpositive, fatherId=fReference[0]}
  [1353] = {x=791.414, y=-152.348, rx=180, rz=148.049, shoulder=lefty, elbow=epositive, wrist=wpositive, fatherId=fReference[0]}
  [1354] = {x=792.709, y=-151.54, rx=180, rz=147.969, shoulder=lefty, elbow=epositive, wrist=wpositive, fatherId=fReference[0]}
  [1355] = {x=794.004, y=-150.73, rx=-180, rz=147.89, shoulder=lefty, elbow=epositive, wrist=wpositive, fatherId=fReference[0]}
  [1356] = {x=795.298, y=-149.918, rx=180, rz=147.811, shoulder=lefty, elbow=epositive, wrist=wpositive, fatherId=fReference[0]}
  [1357] = {x=796.591, y=-149.104, rx=-180, rz=147.733, shoulder=lefty, elbow=epositive, wrist=wpositive, fatherId=fReference[0]}
  [1358] = {x=797.884, y=-148.288, rx=-180, rz=147.656, shoulder=lefty, elbow=epositive, wrist=wpositive, fatherId=fReference[0]}
  [1359] = {x=799.175, y=-147.47, rx=-180, rz=147.579, shoulder=lefty, elbow=epositive, wrist=wpositive, fatherId=fReference[0]}
  [1360] = {x=800.467, y=-146.65, rx=180, rz=147.503, shoulder=lefty, elbow=epositive, wrist=wpositive, fatherId=fReference[0]}
  [1361] = {x=801.757, y=-145.827, rx=180, rz=147.427, shoulder=lefty, elbow=epositive, wrist=wpositive, fatherId=fReference[0]}
  [1362] = {x=803.047, y=-145.003, rx=-180, rz=147.352, shoulder=lefty, elbow=epositive, wrist=wpositive, fatherId=fReference[0]}
  [1363] = {x=804.337, y=-144.177, rx=180, rz=147.277, shoulder=lefty, elbow=epositive, wrist=wpositive, fatherId=fReference[0]}
  [1364] = {x=805.626, y=-143.349, rx=180, rz=147.204, shoulder=lefty, elbow=epositive, wrist=wpositive, fatherId=fReference[0]}
  [1365] = {x=806.914, y=-142.519, rx=-180, rz=147.13, shoulder=lefty, elbow=epositive, wrist=wpositive, fatherId=fReference[0]}
  [1366] = {x=808.201, y=-141.687, rx=-180, rz=147.058, shoulder=lefty, elbow=epositive, wrist=wpositive, fatherId=fReference[0]}
  [1367] = {x=809.488, y=-140.853, rx=-180, rz=146.986, shoulder=lefty, elbow=epositive, wrist=wpositive, fatherId=fReference[0]}
  [1368] = {x=810.774, y=-140.017, rx=180, rz=146.914, shoulder=lefty, elbow=epositive, wrist=wpositive, fatherId=fReference[0]}
  [1369] = {x=812.06, y=-139.18, rx=-180, rz=146.843, shoulder=lefty, elbow=epositive, wrist=wpositive, fatherId=fReference[0]}
  [1370] = {x=813.345, y=-138.34, rx=-180, rz=146.773, shoulder=lefty, elbow=epositive, wrist=wpositive, fatherId=fReference[0]}
  [1371] = {x=814.629, y=-137.499, rx=180, rz=146.703, shoulder=lefty, elbow=epositive, wrist=wpositive, fatherId=fReference[0]}
  [1372] = {x=815.913, y=-136.656, rx=-180, rz=146.634, shoulder=lefty, elbow=epositive, wrist=wpositive, fatherId=fReference[0]}
  [1373] = {x=817.196, y=-135.811, rx=180, rz=146.565, shoulder=lefty, elbow=epositive, wrist=wpositive, fatherId=fReference[0]}
  [1374] = {x=818.479, y=-134.964, rx=180, rz=146.497, shoulder=lefty, elbow=epositive, wrist=wpositive, fatherId=fReference[0]}
  [1375] = {x=819.761, y=-134.115, rx=-180, rz=146.429, shoulder=lefty, elbow=epositive, wrist=wpositive, fatherId=fReference[0]}
  [1376] = {x=821.042, y=-133.265, rx=180, rz=146.362, shoulder=lefty, elbow=epositive, wrist=wpositive, fatherId=fReference[0]}
  [1377] = {x=822.323, y=-132.413, rx=180, rz=146.296, shoulder=lefty, elbow=epositive, wrist=wpositive, fatherId=fReference[0]}
  [1378] = {x=823.603, y=-131.559, rx=-180, rz=146.23, shoulder=lefty, elbow=epositive, wrist=wpositive, fatherId=fReference[0]}
  [1379] = {x=824.882, y=-130.703, rx=180, rz=146.165, shoulder=lefty, elbow=epositive, wrist=wpositive, fatherId=fReference[0]}
  [1380] = {x=826.161, y=-129.846, rx=-180, rz=146.1, shoulder=lefty, elbow=epositive, wrist=wpositive, fatherId=fReference[0]}
  [1381] = {x=827.44, y=-128.987, rx=180, rz=146.036, shoulder=lefty, elbow=epositive, wrist=wpositive, fatherId=fReference[0]}
  [1382] = {x=828.717, y=-128.127, rx=-180, rz=145.972, shoulder=lefty, elbow=epositive, wrist=wpositive, fatherId=fReference[0]}
  [1383] = {x=829.994, y=-127.264, rx=-180, rz=145.909, shoulder=lefty, elbow=epositive, wrist=wpositive, fatherId=fReference[0]}
  [1384] = {x=831.271, y=-126.4, rx=180, rz=145.847, shoulder=lefty, elbow=epositive, wrist=wpositive, fatherId=fReference[0]}
  [1385] = {x=832.547, y=-125.535, rx=-180, rz=145.785, shoulder=lefty, elbow=epositive, wrist=wpositive, fatherId=fReference[0]}
  [1386] = {x=833.822, y=-124.667, rx=180, rz=145.723, shoulder=lefty, elbow=epositive, wrist=wpositive, fatherId=fReference[0]}
  [1387] = {x=835.097, y=-123.798, rx=180, rz=145.662, shoulder=lefty, elbow=epositive, wrist=wpositive, fatherId=fReference[0]}
  [1388] = {x=836.372, y=-122.928, rx=-180, rz=145.602, shoulder=lefty, elbow=epositive, wrist=wpositive, fatherId=fReference[0]}
  [1389] = {x=837.645, y=-122.056, rx=-180, rz=145.542, shoulder=lefty, elbow=epositive, wrist=wpositive, fatherId=fReference[0]}
  [1390] = {x=838.918, y=-121.182, rx=180, rz=145.483, shoulder=lefty, elbow=epositive, wrist=wpositive, fatherId=fReference[0]}
  [1391] = {x=840.191, y=-120.307, rx=-180, rz=145.424, shoulder=lefty, elbow=epositive, wrist=wpositive, fatherId=fReference[0]}
  [1392] = {x=841.463, y=-119.43, rx=-180, rz=145.366, shoulder=lefty, elbow=epositive, wrist=wpositive, fatherId=fReference[0]}
  [1393] = {x=842.734, y=-118.552, rx=180, rz=145.308, shoulder=lefty, elbow=epositive, wrist=wpositive, fatherId=fReference[0]}
  [1394] = {x=844.005, y=-117.672, rx=-180, rz=145.251, shoulder=lefty, elbow=epositive, wrist=wpositive, fatherId=fReference[0]}
  [1395] = {x=845.276, y=-116.791, rx=180, rz=145.195, shoulder=lefty, elbow=epositive, wrist=wpositive, fatherId=fReference[0]}
  [1396] = {x=846.545, y=-115.908, rx=-180, rz=145.139, shoulder=lefty, elbow=epositive, wrist=wpositive, fatherId=fReference[0]}
  [1397] = {x=847.815, y=-115.024, rx=180, rz=145.083, shoulder=lefty, elbow=epositive, wrist=wpositive, fatherId=fReference[0]}
  [1398] = {x=849.084, y=-114.139, rx=-180, rz=145.028, shoulder=lefty, elbow=epositive, wrist=wpositive, fatherId=fReference[0]}
  [1399] = {x=850.352, y=-113.251, rx=180, rz=144.974, shoulder=lefty, elbow=epositive, wrist=wpositive, fatherId=fReference[0]}
  [1400] = {x=851.619, y=-112.363, rx=180, rz=144.92, shoulder=lefty, elbow=epositive, wrist=wpositive, fatherId=fReference[0]}
  [1401] = {x=852.887, y=-111.473, rx=-180, rz=144.866, shoulder=lefty, elbow=epositive, wrist=wpositive, fatherId=fReference[0]}
  [1402] = {x=854.153, y=-110.582, rx=-180, rz=144.813, shoulder=lefty, elbow=epositive, wrist=wpositive, fatherId=fReference[0]}
  [1403] = {x=855.419, y=-109.689, rx=180, rz=144.761, shoulder=lefty, elbow=epositive, wrist=wpositive, fatherId=fReference[0]}
  [1404] = {x=856.685, y=-108.795, rx=-180, rz=144.709, shoulder=lefty, elbow=epositive, wrist=wpositive, fatherId=fReference[0]}
  [1405] = {x=857.95, y=-107.899, rx=180, rz=144.657, shoulder=lefty, elbow=epositive, wrist=wpositive, fatherId=fReference[0]}
  [1406] = {x=859.215, y=-107.003, rx=-180, rz=144.607, shoulder=lefty, elbow=epositive, wrist=wpositive, fatherId=fReference[0]}
  [1407] = {x=860.479, y=-106.104, rx=180, rz=144.556, shoulder=lefty, elbow=epositive, wrist=wpositive, fatherId=fReference[0]}
  [1408] = {x=861.742, y=-105.205, rx=180, rz=144.506, shoulder=lefty, elbow=epositive, wrist=wpositive, fatherId=fReference[0]}
  [1409] = {x=863.006, y=-104.304, rx=180, rz=144.457, shoulder=lefty, elbow=epositive, wrist=wpositive, fatherId=fReference[0]}
  [1410] = {x=864.268, y=-103.402, rx=-180, rz=144.408, shoulder=lefty, elbow=epositive, wrist=wpositive, fatherId=fReference[0]}
  [1411] = {x=865.53, y=-102.499, rx=180, rz=144.36, shoulder=lefty, elbow=epositive, wrist=wpositive, fatherId=fReference[0]}
  [1412] = {x=866.792, y=-101.594, rx=180, rz=144.312, shoulder=lefty, elbow=epositive, wrist=wpositive, fatherId=fReference[0]}
  [1413] = {x=868.053, y=-100.688, rx=-180, rz=144.265, shoulder=lefty, elbow=epositive, wrist=wpositive, fatherId=fReference[0]}
  [1414] = {x=869.314, y=-99.781, rx=-180, rz=144.218, shoulder=lefty, elbow=epositive, wrist=wpositive, fatherId=fReference[0]}
  [1415] = {x=870.574, y=-98.873, rx=180, rz=144.172, shoulder=lefty, elbow=epositive, wrist=wpositive, fatherId=fReference[0]}
  [1416] = {x=871.834, y=-97.963, rx=-180, rz=144.126, shoulder=lefty, elbow=epositive, wrist=wpositive, fatherId=fReference[0]}
  [1417] = {x=873.094, y=-97.052, rx=-180, rz=144.08, shoulder=lefty, elbow=epositive, wrist=wpositive, fatherId=fReference[0]}
  [1418] = {x=874.353, y=-96.14, rx=-180, rz=144.036, shoulder=lefty, elbow=epositive, wrist=wpositive, fatherId=fReference[0]}
  [1419] = {x=875.611, y=-95.227, rx=-180, rz=143.991, shoulder=lefty, elbow=epositive, wrist=wpositive, fatherId=fReference[0]}
  [1420] = {x=876.869, y=-94.313, rx=-180, rz=143.947, shoulder=lefty, elbow=epositive, wrist=wpositive, fatherId=fReference[0]}
  [1421] = {x=878.127, y=-93.397, rx=180, rz=143.904, shoulder=lefty, elbow=epositive, wrist=wpositive, fatherId=fReference[0]}
  [1422] = {x=879.384, y=-92.481, rx=-180, rz=143.861, shoulder=lefty, elbow=epositive, wrist=wpositive, fatherId=fReference[0]}
  [1423] = {x=880.641, y=-91.563, rx=-180, rz=143.819, shoulder=lefty, elbow=epositive, wrist=wpositive, fatherId=fReference[0]}
  [1424] = {x=881.897, y=-90.644, rx=-180, rz=143.777, shoulder=lefty, elbow=epositive, wrist=wpositive, fatherId=fReference[0]}
  [1425] = {x=883.153, y=-89.724, rx=180, rz=143.735, shoulder=lefty, elbow=epositive, wrist=wpositive, fatherId=fReference[0]}
  [1426] = {x=884.409, y=-88.803, rx=180, rz=143.694, shoulder=lefty, elbow=epositive, wrist=wpositive, fatherId=fReference[0]}
  [1427] = {x=885.664, y=-87.881, rx=-180, rz=143.654, shoulder=lefty, elbow=epositive, wrist=wpositive, fatherId=fReference[0]}
  [1428] = {x=886.919, y=-86.957, rx=180, rz=143.614, shoulder=lefty, elbow=epositive, wrist=wpositive, fatherId=fReference[0]}
  [1429] = {x=888.173, y=-86.033, rx=-180, rz=143.574, shoulder=lefty, elbow=epositive, wrist=wpositive, fatherId=fReference[0]}
  [1430] = {x=889.427, y=-85.108, rx=-180, rz=143.535, shoulder=lefty, elbow=epositive, wrist=wpositive, fatherId=fReference[0]}
  [1431] = {x=890.681, y=-84.181, rx=180, rz=143.497, shoulder=lefty, elbow=epositive, wrist=wpositive, fatherId=fReference[0]}
  [1432] = {x=891.934, y=-83.254, rx=-180, rz=143.459, shoulder=lefty, elbow=epositive, wrist=wpositive, fatherId=fReference[0]}
  [1433] = {x=893.187, y=-82.325, rx=180, rz=143.421, shoulder=lefty, elbow=epositive, wrist=wpositive, fatherId=fReference[0]}
  [1434] = {x=894.439, y=-81.396, rx=-180, rz=143.384, shoulder=lefty, elbow=epositive, wrist=wpositive, fatherId=fReference[0]}
  [1435] = {x=895.691, y=-80.465, rx=180, rz=143.347, shoulder=lefty, elbow=epositive, wrist=wpositive, fatherId=fReference[0]}
  [1436] = {x=896.943, y=-79.534, rx=-180, rz=143.311, shoulder=lefty, elbow=epositive, wrist=wpositive, fatherId=fReference[0]}
  [1437] = {x=898.195, y=-78.602, rx=180, rz=143.275, shoulder=lefty, elbow=epositive, wrist=wpositive, fatherId=fReference[0]}
  [1438] = {x=899.446, y=-77.668, rx=180, rz=143.24, shoulder=lefty, elbow=epositive, wrist=wpositive, fatherId=fReference[0]}
  [1439] = {x=900.696, y=-76.734, rx=-180, rz=143.205, shoulder=lefty, elbow=epositive, wrist=wpositive, fatherId=fReference[0]}
  [1440] = {x=901.947, y=-75.799, rx=180, rz=143.171, shoulder=lefty, elbow=epositive, wrist=wpositive, fatherId=fReference[0]}
  [1441] = {x=903.197, y=-74.862, rx=-180, rz=143.137, shoulder=lefty, elbow=epositive, wrist=wpositive, fatherId=fReference[0]}
  [1442] = {x=904.447, y=-73.925, rx=180, rz=143.103, shoulder=lefty, elbow=epositive, wrist=wpositive, fatherId=fReference[0]}
  [1443] = {x=905.696, y=-72.987, rx=-180, rz=143.07, shoulder=lefty, elbow=epositive, wrist=wpositive, fatherId=fReference[0]}
  [1444] = {x=906.945, y=-72.049, rx=180, rz=143.038, shoulder=lefty, elbow=epositive, wrist=wpositive, fatherId=fReference[0]}
  [1445] = {x=908.194, y=-71.109, rx=180, rz=143.006, shoulder=lefty, elbow=epositive, wrist=wpositive, fatherId=fReference[0]}
  [1446] = {x=909.442, y=-70.168, rx=180, rz=142.974, shoulder=lefty, elbow=epositive, wrist=wpositive, fatherId=fReference[0]}
  [1447] = {x=910.69, y=-69.227, rx=180, rz=142.943, shoulder=lefty, elbow=epositive, wrist=wpositive, fatherId=fReference[0]}
  [1448] = {x=911.938, y=-68.285, rx=180, rz=142.912, shoulder=lefty, elbow=epositive, wrist=wpositive, fatherId=fReference[0]}
  [1449] = {x=913.185, y=-67.342, rx=180, rz=142.882, shoulder=lefty, elbow=epositive, wrist=wpositive, fatherId=fReference[0]}
  [1450] = {x=914.433, y=-66.398, rx=180, rz=142.853, shoulder=lefty, elbow=epositive, wrist=wpositive, fatherId=fReference[0]}
  [1451] = {x=915.68, y=-65.453, rx=180, rz=142.823, shoulder=lefty, elbow=epositive, wrist=wpositive, fatherId=fReference[0]}
  [1452] = {x=916.926, y=-64.508, rx=180, rz=142.794, shoulder=lefty, elbow=epositive, wrist=wpositive, fatherId=fReference[0]}
  [1453] = {x=918.172, y=-63.562, rx=180, rz=142.766, shoulder=lefty, elbow=epositive, wrist=wpositive, fatherId=fReference[0]}
  [1454] = {x=919.418, y=-62.615, rx=-180, rz=142.738, shoulder=lefty, elbow=epositive, wrist=wpositive, fatherId=fReference[0]}
  [1455] = {x=920.664, y=-61.667, rx=-180, rz=142.71, shoulder=lefty, elbow=epositive, wrist=wpositive, fatherId=fReference[0]}
  [1456] = {x=921.91, y=-60.719, rx=180, rz=142.683, shoulder=lefty, elbow=epositive, wrist=wpositive, fatherId=fReference[0]}
  [1457] = {x=923.155, y=-59.769, rx=180, rz=142.657, shoulder=lefty, elbow=epositive, wrist=wpositive, fatherId=fReference[0]}
  [1458] = {x=924.4, y=-58.82, rx=180, rz=142.631, shoulder=lefty, elbow=epositive, wrist=wpositive, fatherId=fReference[0]}
  [1459] = {x=925.644, y=-57.869, rx=-180, rz=142.605, shoulder=lefty, elbow=epositive, wrist=wpositive, fatherId=fReference[0]}
  [1460] = {x=926.889, y=-56.918, rx=180, rz=142.58, shoulder=lefty, elbow=epositive, wrist=wpositive, fatherId=fReference[0]}
  [1461] = {x=928.133, y=-55.966, rx=180, rz=142.555, shoulder=lefty, elbow=epositive, wrist=wpositive, fatherId=fReference[0]}
  [1462] = {x=929.377, y=-55.013, rx=-180, rz=142.53, shoulder=lefty, elbow=epositive, wrist=wpositive, fatherId=fReference[0]}
  [1463] = {x=930.621, y=-54.06, rx=180, rz=142.507, shoulder=lefty, elbow=epositive, wrist=wpositive, fatherId=fReference[0]}
  [1464] = {x=931.864, y=-53.106, rx=180, rz=142.483, shoulder=lefty, elbow=epositive, wrist=wpositive, fatherId=fReference[0]}
  [1465] = {x=933.107, y=-52.152, rx=180, rz=142.46, shoulder=lefty, elbow=epositive, wrist=wpositive, fatherId=fReference[0]}
  [1466] = {x=934.35, y=-51.197, rx=-180, rz=142.437, shoulder=lefty, elbow=epositive, wrist=wpositive, fatherId=fReference[0]}
  [1467] = {x=935.593, y=-50.241, rx=-180, rz=142.415, shoulder=lefty, elbow=epositive, wrist=wpositive, fatherId=fReference[0]}
  [1468] = {x=936.835, y=-49.284, rx=-180, rz=142.393, shoulder=lefty, elbow=epositive, wrist=wpositive, fatherId=fReference[0]}
  [1469] = {x=938.078, y=-48.328, rx=180, rz=142.372, shoulder=lefty, elbow=epositive, wrist=wpositive, fatherId=fReference[0]}
  [1470] = {x=939.32, y=-47.37, rx=-180, rz=142.351, shoulder=lefty, elbow=epositive, wrist=wpositive, fatherId=fReference[0]}
  [1471] = {x=940.561, y=-46.412, rx=180, rz=142.331, shoulder=lefty, elbow=epositive, wrist=wpositive, fatherId=fReference[0]}
  [1472] = {x=941.803, y=-45.454, rx=180, rz=142.311, shoulder=lefty, elbow=epositive, wrist=wpositive, fatherId=fReference[0]}
  [1473] = {x=943.044, y=-44.494, rx=180, rz=142.291, shoulder=lefty, elbow=epositive, wrist=wpositive, fatherId=fReference[0]}
  [1474] = {x=944.286, y=-43.535, rx=-180, rz=142.272, shoulder=lefty, elbow=epositive, wrist=wpositive, fatherId=fReference[0]}
  [1475] = {x=945.527, y=-42.575, rx=180, rz=142.254, shoulder=lefty, elbow=epositive, wrist=wpositive, fatherId=fReference[0]}
  [1476] = {x=946.768, y=-41.614, rx=180, rz=142.235, shoulder=lefty, elbow=epositive, wrist=wpositive, fatherId=fReference[0]}
  [1477] = {x=948.008, y=-40.653, rx=180, rz=142.217, shoulder=lefty, elbow=epositive, wrist=wpositive, fatherId=fReference[0]}
  [1478] = {x=949.249, y=-39.691, rx=180, rz=142.2, shoulder=lefty, elbow=epositive, wrist=wpositive, fatherId=fReference[0]}
  [1479] = {x=950.489, y=-38.729, rx=180, rz=142.183, shoulder=lefty, elbow=epositive, wrist=wpositive, fatherId=fReference[0]}
  [1480] = {x=951.729, y=-37.767, rx=-180, rz=142.167, shoulder=lefty, elbow=epositive, wrist=wpositive, fatherId=fReference[0]}
  [1481] = {x=952.969, y=-36.804, rx=180, rz=142.151, shoulder=lefty, elbow=epositive, wrist=wpositive, fatherId=fReference[0]}
  [1482] = {x=954.209, y=-35.841, rx=180, rz=142.135, shoulder=lefty, elbow=epositive, wrist=wpositive, fatherId=fReference[0]}
  [1483] = {x=955.448, y=-34.877, rx=180, rz=142.12, shoulder=lefty, elbow=epositive, wrist=wpositive, fatherId=fReference[0]}
  [1484] = {x=956.688, y=-33.913, rx=180, rz=142.105, shoulder=lefty, elbow=epositive, wrist=wpositive, fatherId=fReference[0]}
  [1485] = {x=957.927, y=-32.948, rx=180, rz=142.09, shoulder=lefty, elbow=epositive, wrist=wpositive, fatherId=fReference[0]}
  [1486] = {x=959.166, y=-31.983, rx=180, rz=142.076, shoulder=lefty, elbow=epositive, wrist=wpositive, fatherId=fReference[0]}
  [1487] = {x=960.405, y=-31.018, rx=-180, rz=142.063, shoulder=lefty, elbow=epositive, wrist=wpositive, fatherId=fReference[0]}
  [1488] = {x=961.644, y=-30.052, rx=-180, rz=142.05, shoulder=lefty, elbow=epositive, wrist=wpositive, fatherId=fReference[0]}
  [1489] = {x=962.882, y=-29.086, rx=180, rz=142.037, shoulder=lefty, elbow=epositive, wrist=wpositive, fatherId=fReference[0]}
  [1490] = {x=964.121, y=-28.12, rx=-180, rz=142.025, shoulder=lefty, elbow=epositive, wrist=wpositive, fatherId=fReference[0]}
  [1491] = {x=965.359, y=-27.153, rx=180, rz=142.013, shoulder=lefty, elbow=epositive, wrist=wpositive, fatherId=fReference[0]}
  [1492] = {x=966.598, y=-26.186, rx=-180, rz=142.002, shoulder=lefty, elbow=epositive, wrist=wpositive, fatherId=fReference[0]}
  [1493] = {x=967.836, y=-25.219, rx=180, rz=141.991, shoulder=lefty, elbow=epositive, wrist=wpositive, fatherId=fReference[0]}
  [1494] = {x=969.074, y=-24.251, rx=-180, rz=141.98, shoulder=lefty, elbow=epositive, wrist=wpositive, fatherId=fReference[0]}
  [1495] = {x=970.312, y=-23.283, rx=180, rz=141.97, shoulder=lefty, elbow=epositive, wrist=wpositive, fatherId=fReference[0]}
  [1496] = {x=971.55, y=-22.315, rx=180, rz=141.96, shoulder=lefty, elbow=epositive, wrist=wpositive, fatherId=fReference[0]}
  [1497] = {x=972.787, y=-21.347, rx=180, rz=141.951, shoulder=lefty, elbow=epositive, wrist=wpositive, fatherId=fReference[0]}
  [1498] = {x=974.025, y=-20.378, rx=-180, rz=141.942, shoulder=lefty, elbow=epositive, wrist=wpositive, fatherId=fReference[0]}
  [1499] = {x=975.263, y=-19.409, rx=180, rz=141.934, shoulder=lefty, elbow=epositive, wrist=wpositive, fatherId=fReference[0]}
  [1500] = {x=976.5, y=-18.44, rx=-180, rz=141.926, shoulder=lefty, elbow=epositive, wrist=wpositive, fatherId=fReference[0]}
  [1501] = {x=977.737, y=-17.471, rx=180, rz=141.918, shoulder=lefty, elbow=epositive, wrist=wpositive, fatherId=fReference[0]}
  [1502] = {x=978.975, y=-16.501, rx=180, rz=141.911, shoulder=lefty, elbow=epositive, wrist=wpositive, fatherId=fReference[0]}
  [1503] = {x=980.212, y=-15.532, rx=180, rz=141.904, shoulder=lefty, elbow=epositive, wrist=wpositive, fatherId=fReference[0]}
  [1504] = {x=981.449, y=-14.562, rx=-180, rz=141.898, shoulder=lefty, elbow=epositive, wrist=wpositive, fatherId=fReference[0]}
  [1505] = {x=982.686, y=-13.592, rx=180, rz=141.892, shoulder=lefty, elbow=epositive, wrist=wpositive, fatherId=fReference[0]}
  [1506] = {x=983.923, y=-12.621, rx=180, rz=141.887, shoulder=lefty, elbow=epositive, wrist=wpositive, fatherId=fReference[0]}
  [1507] = {x=985.16, y=-11.651, rx=-180, rz=141.882, shoulder=lefty, elbow=epositive, wrist=wpositive, fatherId=fReference[0]}
  [1508] = {x=986.397, y=-10.681, rx=180, rz=141.877, shoulder=lefty, elbow=epositive, wrist=wpositive, fatherId=fReference[0]}
  [1509] = {x=987.634, y=-9.71, rx=180, rz=141.873, shoulder=lefty, elbow=epositive, wrist=wpositive, fatherId=fReference[0]}
  [1510] = {x=988.87, y=-8.739, rx=180, rz=141.869, shoulder=lefty, elbow=epositive, wrist=wpositive, fatherId=fReference[0]}
  [1511] = {x=990.107, y=-7.769, rx=-180, rz=141.866, shoulder=lefty, elbow=epositive, wrist=wpositive, fatherId=fReference[0]}
  [1512] = {x=991.344, y=-6.798, rx=180, rz=141.863, shoulder=lefty, elbow=epositive, wrist=wpositive, fatherId=fReference[0]}
  [1513] = {x=992.58, y=-5.827, rx=-180, rz=141.86, shoulder=lefty, elbow=epositive, wrist=wpositive, fatherId=fReference[0]}
  [1514] = {x=993.817, y=-4.856, rx=180, rz=141.858, shoulder=lefty, elbow=epositive, wrist=wpositive, fatherId=fReference[0]}
  [1515] = {x=995.054, y=-3.885, rx=180, rz=141.857, shoulder=lefty, elbow=epositive, wrist=wpositive, fatherId=fReference[0]}
  [1516] = {x=996.29, y=-2.914, rx=-180, rz=141.855, shoulder=lefty, elbow=epositive, wrist=wpositive, fatherId=fReference[0]}
  [1517] = {x=997.527, y=-1.942, rx=180, rz=141.854, shoulder=lefty, elbow=epositive, wrist=wpositive, fatherId=fReference[0]}
  [1518] = {x=998.763, y=-0.971, rx=-180, rz=141.854, shoulder=lefty, elbow=epositive, wrist=wpositive, fatherId=fReference[0]}
  [1519] = {x=1000, rx=180, rz=141.854, shoulder=lefty, elbow=epositive, wrist=wpositive, fatherId=fReference[0]}
  [1520] = {x=1000, rx=180, rz=141.854, shoulder=lefty, elbow=epositive, wrist=wpositive, fatherId=fReference[0]}
  [1521] = {x=1000, z=100, rx=180, rz=141.854, shoulder=lefty, elbow=epositive, wrist=wpositive, fatherId=fReference[0]}
  [1522] = {x=-1000, z=122, rx=180, rz=141.854, shoulder=lefty, elbow=epositive, wrist=wpositive, fatherId=fReference[0]}
  [1523] = {x=-1000, z=22, rx=180, rz=141.854, shoulder=lefty, elbow=epositive, wrist=wpositive, fatherId=fReference[0]}
  [1524] = {x=-1000, z=22, rx=180, rz=141.854, shoulder=lefty, elbow=epositive, wrist=wpositive, fatherId=fReference[0]}
  [1525] = {x=-998.763, y=0.971, z=22, rx=180, rz=141.854, shoulder=lefty, elbow=epositive, wrist=wpositive, fatherId=fReference[0]}
  [1526] = {x=-997.527, y=1.942, z=22, rx=180, rz=141.855, shoulder=lefty, elbow=epositive, wrist=wpositive, fatherId=fReference[0]}
  [1527] = {x=-996.29, y=2.914, z=22, rx=180, rz=141.857, shoulder=lefty, elbow=epositive, wrist=wpositive, fatherId=fReference[0]}
  [1528] = {x=-995.054, y=3.885, z=22, rx=180, rz=141.858, shoulder=lefty, elbow=epositive, wrist=wpositive, fatherId=fReference[0]}
  [1529] = {x=-993.817, y=4.856, z=22, rx=180, rz=141.86, shoulder=lefty, elbow=epositive, wrist=wpositive, fatherId=fReference[0]}
  [1530] = {x=-992.58, y=5.827, z=22, rx=180, rz=141.863, shoulder=lefty, elbow=epositive, wrist=wpositive, fatherId=fReference[0]}
  [1531] = {x=-991.344, y=6.798, z=22, rx=180, rz=141.866, shoulder=lefty, elbow=epositive, wrist=wpositive, fatherId=fReference[0]}
  [1532] = {x=-990.107, y=7.769, z=22, rx=180, rz=141.869, shoulder=lefty, elbow=epositive, wrist=wpositive, fatherId=fReference[0]}
  [1533] = {x=-988.87, y=8.739, z=22, rx=180, rz=141.873, shoulder=lefty, elbow=epositive, wrist=wpositive, fatherId=fReference[0]}
  [1534] = {x=-987.634, y=9.71, z=22, rx=180, rz=141.877, shoulder=lefty, elbow=epositive, wrist=wpositive, fatherId=fReference[0]}
  [1535] = {x=-986.397, y=10.681, z=22, rx=180, rz=141.882, shoulder=lefty, elbow=epositive, wrist=wpositive, fatherId=fReference[0]}
  [1536] = {x=-985.16, y=11.651, z=22, rx=180, rz=141.887, shoulder=lefty, elbow=epositive, wrist=wpositive, fatherId=fReference[0]}
  [1537] = {x=-983.923, y=12.622, z=22, rx=180, rz=141.892, shoulder=lefty, elbow=epositive, wrist=wpositive, fatherId=fReference[0]}
  [1538] = {x=-982.686, y=13.592, z=22, rx=180, rz=141.898, shoulder=lefty, elbow=epositive, wrist=wpositive, fatherId=fReference[0]}
  [1539] = {x=-981.449, y=14.562, z=22, rx=180, rz=141.904, shoulder=lefty, elbow=epositive, wrist=wpositive, fatherId=fReference[0]}
  [1540] = {x=-980.211, y=15.532, z=22, rx=180, rz=141.911, shoulder=lefty, elbow=epositive, wrist=wpositive, fatherId=fReference[0]}
  [1541] = {x=-978.974, y=16.502, z=22, rx=180, rz=141.918, shoulder=lefty, elbow=epositive, wrist=wpositive, fatherId=fReference[0]}
  [1542] = {x=-977.737, y=17.471, z=22, rx=180, rz=141.926, shoulder=lefty, elbow=epositive, wrist=wpositive, fatherId=fReference[0]}
  [1543] = {x=-976.499, y=18.441, z=22, rx=180, rz=141.934, shoulder=lefty, elbow=epositive, wrist=wpositive, fatherId=fReference[0]}
  [1544] = {x=-975.262, y=19.41, z=22, rx=180, rz=141.942, shoulder=lefty, elbow=epositive, wrist=wpositive, fatherId=fReference[0]}
  [1545] = {x=-974.024, y=20.379, z=22, rx=180, rz=141.951, shoulder=lefty, elbow=epositive, wrist=wpositive, fatherId=fReference[0]}
  [1546] = {x=-972.786, y=21.347, z=22, rx=180, rz=141.96, shoulder=lefty, elbow=epositive, wrist=wpositive, fatherId=fReference[0]}
  [1547] = {x=-971.549, y=22.316, z=22, rx=180, rz=141.97, shoulder=lefty, elbow=epositive, wrist=wpositive, fatherId=fReference[0]}
  [1548] = {x=-970.311, y=23.284, z=22, rx=180, rz=141.98, shoulder=lefty, elbow=epositive, wrist=wpositive, fatherId=fReference[0]}
  [1549] = {x=-969.072, y=24.252, z=22, rx=180, rz=141.991, shoulder=lefty, elbow=epositive, wrist=wpositive, fatherId=fReference[0]}
  [1550] = {x=-967.834, y=25.22, z=22, rx=180, rz=142.002, shoulder=lefty, elbow=epositive, wrist=wpositive, fatherId=fReference[0]}
  [1551] = {x=-966.596, y=26.187, z=22, rx=180, rz=142.013, shoulder=lefty, elbow=epositive, wrist=wpositive, fatherId=fReference[0]}
  [1552] = {x=-965.357, y=27.155, z=22, rx=180, rz=142.025, shoulder=lefty, elbow=epositive, wrist=wpositive, fatherId=fReference[0]}
